Yaskawa INFORM job: apremTRJ4.JBI

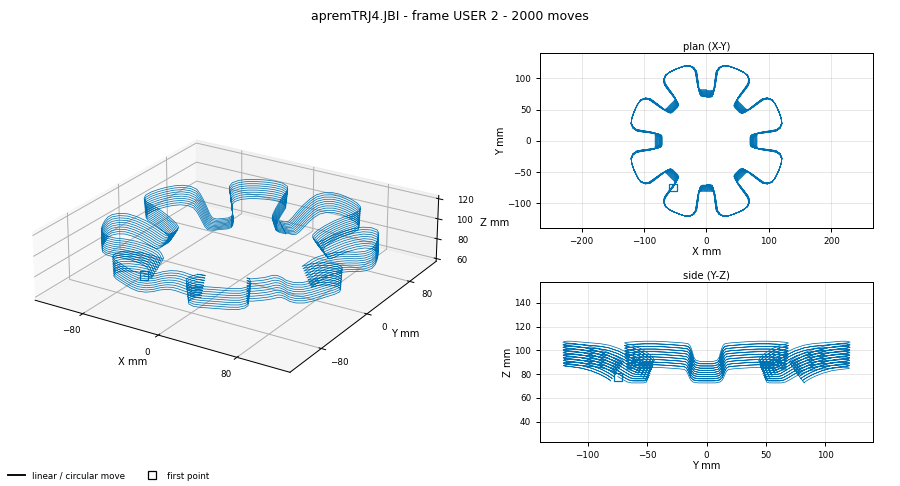
[picture p0: tool path of apremTRJ4.JBI in frame USER 2, 2000 of 2000 moves have a stored position in this frame; points joined in program order, loops and branches not executed]
/JOB
//NAME apremTRJ4
//POS
///NPOS 2000,0,0,0,0,0
///USER 2
///TOOL 1
///POSTYPE USER
///RECTAN
///RCONF 1,0,0,0,0,0,0,0,0,0,0,0,0,0,0,0,0,0,0,0,0,0,0,0
C00000=-53.765,-74.632,78.012,177.9395,-3.2342,0.0000
C00001=-51.010,-70.134,75.345,-179.2635,1.4013,0.0000
C00002=-50.421,-66.568,73.433,174.4013,27.1844,0.0000
C00003=-52.955,-63.098,72.678,152.6245,29.3823,0.0000
C00004=-55.786,-60.507,72.646,149.9913,27.7136,0.0000
C00005=-58.192,-58.192,72.667,151.1075,28.8919,0.0000
C00006=-60.507,-55.786,72.646,152.2867,30.0091,0.0000
C00007=-63.099,-52.955,72.678,150.6167,27.3735,0.0000
C00008=-66.568,-50.421,73.433,152.8156,5.5988,0.0000
C00009=-70.134,-51.010,75.345,178.5987,-0.7365,0.0000
C00010=-74.632,-53.765,78.012,-176.7658,2.0605,0.0000
C00011=-80.322,-57.816,80.784,-174.8040,3.4978,0.0000
C00012=-86.699,-62.416,82.923,-173.5056,4.3301,0.0000
C00013=-92.902,-66.405,83.982,-172.7331,2.9843,0.0000
C00014=-99.586,-67.141,84.541,-175.1721,-0.8383,0.0000
C00015=-105.834,-64.370,84.996,-178.0904,-1.4950,0.0000
C00016=-110.354,-58.600,85.456,-179.9251,-0.1383,0.0000
C00017=-113.876,-51.533,85.759,-179.9922,-0.0171,0.0000
C00018=-116.962,-44.084,85.759,-179.9934,-0.0176,0.0000
C00019=-119.469,-36.595,85.456,-179.9552,-0.1508,0.0000
C00020=-120.352,-29.319,84.996,179.7066,-2.4067,0.0000
C00021=-117.894,-22.942,84.541,177.1732,-4.0082,0.0000
C00022=-112.647,-18.736,83.982,172.7605,-3.0512,0.0000
C00023=-105.440,-17.170,82.923,172.3659,-1.5439,0.0000
C00024=-97.679,-15.914,80.784,173.8630,-1.2077,0.0000
C00025=-90.790,-14.755,78.012,176.2584,-0.8317,0.0000
C00026=-85.662,-13.522,75.345,-178.4885,0.4702,0.0000
C00027=-82.723,-11.418,73.433,-163.6249,23.3873,0.0000
C00028=-82.062,-7.172,72.678,-178.1671,37.3904,0.0000
C00029=-82.232,-3.338,72.646,177.8846,37.9487,0.0000
C00030=-82.296,0.000,72.667,179.9994,37.9698,0.0000
C00031=-82.232,3.338,72.646,-177.8840,37.9488,0.0000
C00032=-82.062,7.172,72.678,178.1644,37.3898,0.0000
C00033=-82.723,11.418,73.433,163.6250,23.3874,0.0000
C00034=-85.662,13.522,75.345,178.4885,0.4702,0.0000
C00035=-90.790,14.755,78.012,-176.2584,-0.8317,0.0000
C00036=-97.679,15.914,80.784,-173.8630,-1.2077,0.0000
C00037=-105.440,17.170,82.923,-172.3659,-1.5439,0.0000
C00038=-112.647,18.736,83.982,-172.7605,-3.0512,0.0000
C00039=-117.894,22.942,84.541,-177.1732,-4.0082,0.0000
C00040=-120.352,29.319,84.996,-179.7066,-2.4067,0.0000
C00041=-119.469,36.595,85.456,179.9552,-0.1508,0.0000
C00042=-116.962,44.084,85.759,179.9934,-0.0176,0.0000
C00043=-113.876,51.533,85.759,179.9922,-0.0171,0.0000
C00044=-110.354,58.600,85.456,179.9251,-0.1383,0.0000
C00045=-105.834,64.370,84.996,178.0904,-1.4950,0.0000
C00046=-99.586,67.141,84.541,175.1721,-0.8383,0.0000
C00047=-92.902,66.405,83.982,172.7331,2.9843,0.0000
C00048=-86.699,62.416,82.923,173.5056,4.3301,0.0000
C00049=-80.322,57.816,80.784,174.8040,3.4978,0.0000
C00050=-74.632,53.765,78.012,176.7658,2.0605,0.0000
C00051=-70.134,51.010,75.345,-178.5987,-0.7365,0.0000
C00052=-66.568,50.421,73.433,-152.8156,5.5987,0.0000
C00053=-63.098,52.955,72.678,-150.6177,27.3755,0.0000
C00054=-60.507,55.786,72.646,-152.2864,30.0087,0.0000
C00055=-58.192,58.192,72.667,-151.1081,28.8925,0.0000
C00056=-55.786,60.507,72.646,-149.9909,27.7133,0.0000
C00057=-52.955,63.099,72.678,-152.6265,29.3833,0.0000
C00058=-50.421,66.568,73.433,-174.4012,27.1844,0.0000
C00059=-51.010,70.134,75.345,179.2635,1.4013,0.0000
C00060=-53.765,74.632,78.012,-177.9395,-3.2342,0.0000
C00061=-57.816,80.322,80.784,-176.5022,-5.1960,0.0000
C00062=-62.416,86.699,82.923,-175.6699,-6.4944,0.0000
C00063=-66.405,92.902,83.982,-177.0157,-7.2669,0.0000
C00064=-67.141,99.586,84.541,179.1617,-4.8279,0.0000
C00065=-64.370,105.834,84.996,178.5050,-1.9096,0.0000
C00066=-58.600,110.354,85.456,179.8617,-0.0749,0.0000
C00067=-51.533,113.876,85.759,179.9829,-0.0078,0.0000
C00068=-44.084,116.962,85.759,179.9824,-0.0066,0.0000
C00069=-36.595,119.469,85.456,179.8492,-0.0448,0.0000
C00070=-29.319,120.352,84.996,177.5933,0.2934,0.0000
C00071=-22.942,117.894,84.541,175.9918,2.8268,0.0000
C00072=-18.736,112.647,83.982,176.9488,7.2395,0.0000
C00073=-17.170,105.440,82.923,178.4561,7.6341,0.0000
C00074=-15.914,97.679,80.784,178.7923,6.1370,0.0000
C00075=-14.755,90.790,78.012,179.1683,3.7416,0.0000
C00076=-13.522,85.662,75.345,-179.5298,-1.5115,0.0000
C00077=-11.418,82.723,73.433,-156.6126,-16.3750,0.0000
C00078=-7.172,82.062,72.678,-142.6102,-1.8356,0.0000
C00079=-3.338,82.232,72.646,-142.0512,2.1160,0.0000
C00080=0.000,82.296,72.667,-142.0302,-0.0006,0.0000
C00081=0.000,80.948,74.406,-142.4252,-0.0006,0.0000
C00082=3.215,80.888,74.384,-142.4452,-2.0536,0.0000
C00083=6.965,80.731,74.417,-143.0509,2.1075,0.0000
C00084=11.165,81.441,75.203,-157.7434,16.2795,0.0000
C00085=13.215,84.505,77.191,-179.7323,0.9131,0.0000
C00086=14.409,89.830,79.960,179.1649,-3.9269,0.0000
C00087=15.548,96.964,82.833,178.8415,-6.1204,0.0000
C00088=16.788,104.985,85.041,178.5474,-7.5066,0.0000
C00089=18.327,112.424,86.132,177.1014,-7.1283,0.0000
C00090=22.561,117.848,86.707,176.0893,-2.8270,0.0000
C00091=29.019,120.407,87.175,177.6414,-0.3022,0.0000
C00092=36.407,119.531,87.647,179.8514,0.0441,0.0000
C00093=44.020,116.986,87.958,179.9827,0.0065,0.0000
C00094=51.595,113.849,87.958,179.9832,0.0077,0.0000
C00095=58.777,110.265,87.647,179.8638,0.0739,0.0000
C00096=64.621,105.660,87.175,178.5453,1.8817,0.0000
C00097=67.378,99.284,86.707,179.2311,4.7592,0.0000
C00098=66.537,92.455,86.132,-176.9875,7.0817,0.0000
C00099=62.365,86.107,85.041,-175.6969,6.3399,0.0000
C00100=57.570,79.558,82.833,-176.4794,5.1497,0.0000
C00101=53.330,73.708,79.960,-177.8105,3.3677,0.0000
C00102=50.409,69.099,77.191,179.5436,-0.8349,0.0000
C00103=49.693,65.482,75.203,-175.2620,-26.3759,0.0000
C00104=52.161,62.011,74.417,-153.1680,-29.1562,0.0000
C00105=54.923,59.470,74.384,-150.3596,-27.3978,0.0000
C00106=57.239,57.239,74.406,-151.4512,-28.5481,0.0000
C00107=59.470,54.923,74.384,-152.6025,-29.6408,0.0000
C00108=62.011,52.160,74.417,-150.8427,-26.8300,0.0000
C00109=65.482,49.693,75.203,-153.6242,-4.7380,0.0000
C00110=69.099,50.409,77.191,-179.1651,0.4564,0.0000
C00111=73.708,53.330,79.960,176.6323,-2.1895,0.0000
C00112=79.558,57.570,82.833,174.8503,-3.5206,0.0000
C00113=86.107,62.365,85.041,173.6601,-4.3031,0.0000
C00114=92.455,66.537,86.132,172.9183,-3.0125,0.0000
C00115=99.284,67.378,86.707,175.2408,0.7689,0.0000
C00116=105.660,64.621,87.175,178.1183,1.4547,0.0000
C00117=110.265,58.777,87.647,179.9261,0.1362,0.0000
C00118=113.849,51.595,87.958,179.9923,0.0168,0.0000
C00119=116.986,44.020,87.958,179.9935,0.0173,0.0000
C00120=119.531,36.407,87.647,179.9559,0.1486,0.0000
C00121=120.407,29.019,87.175,-179.6978,2.3586,0.0000
C00122=117.848,22.561,86.707,-177.1730,3.9107,0.0000
C00123=112.424,18.327,86.132,-172.8717,2.8986,0.0000
C00124=104.985,16.788,85.041,-172.4934,1.4526,0.0000
C00125=96.964,15.548,82.833,-173.8796,1.1585,0.0000
C00126=89.830,14.409,79.960,-176.0731,0.8351,0.0000
C00127=84.505,13.215,77.191,179.0869,-0.2677,0.0000
C00128=81.441,11.165,75.203,163.7205,-22.2566,0.0000
C00129=80.731,6.965,74.417,177.8925,-36.9491,0.0000
C00130=80.888,3.215,74.384,-177.9464,-37.5548,0.0000
C00131=80.948,0.000,74.406,-179.9994,-37.5748,0.0000
C00132=80.888,-3.215,74.384,177.9457,-37.5548,0.0000
C00133=80.731,-6.965,74.417,-177.8898,-36.9485,0.0000
C00134=81.441,-11.165,75.203,-163.7205,-22.2566,0.0000
C00135=84.505,-13.215,77.191,-179.0869,-0.2677,0.0000
C00136=89.830,-14.409,79.960,176.0731,0.8351,0.0000
C00137=96.964,-15.548,82.833,173.8796,1.1585,0.0000
C00138=104.985,-16.788,85.041,172.4934,1.4526,0.0000
C00139=112.424,-18.327,86.132,172.8717,2.8986,0.0000
C00140=117.848,-22.561,86.707,177.1730,3.9107,0.0000
C00141=120.407,-29.019,87.175,179.6978,2.3586,0.0000
C00142=119.531,-36.407,87.647,-179.9559,0.1486,0.0000
C00143=116.986,-44.020,87.958,-179.9935,0.0173,0.0000
C00144=113.849,-51.595,87.958,-179.9923,0.0168,0.0000
C00145=110.265,-58.777,87.647,-179.9261,0.1362,0.0000
C00146=105.660,-64.621,87.175,-178.1183,1.4547,0.0000
C00147=99.284,-67.378,86.707,-175.2408,0.7689,0.0000
C00148=92.455,-66.537,86.132,-172.9183,-3.0125,0.0000
C00149=86.107,-62.365,85.041,-173.6601,-4.3031,0.0000
C00150=79.558,-57.570,82.833,-174.8503,-3.5206,0.0000
C00151=73.708,-53.330,79.960,-176.6323,-2.1895,0.0000
C00152=69.099,-50.409,77.191,179.1651,0.4564,0.0000
C00153=65.482,-49.693,75.203,153.6241,-4.7380,0.0000
C00154=62.011,-52.161,74.417,150.8438,-26.8320,0.0000
C00155=59.470,-54.923,74.384,152.6022,-29.6404,0.0000
C00156=57.239,-57.239,74.406,151.4519,-28.5488,0.0000
C00157=54.923,-59.470,74.384,150.3592,-27.3975,0.0000
C00158=52.160,-62.011,74.417,153.1700,-29.1573,0.0000
C00159=49.693,-65.482,75.203,175.2620,-26.3758,0.0000
C00160=50.409,-69.099,77.191,-179.5436,-0.8349,0.0000
C00161=53.330,-73.708,79.960,177.8105,3.3677,0.0000
C00162=57.570,-79.558,82.833,176.4794,5.1497,0.0000
C00163=62.365,-86.107,85.041,175.6969,6.3399,0.0000
C00164=66.537,-92.455,86.132,176.9875,7.0817,0.0000
C00165=67.378,-99.284,86.707,-179.2311,4.7592,0.0000
C00166=64.621,-105.660,87.175,-178.5453,1.8817,0.0000
C00167=58.777,-110.265,87.647,-179.8638,0.0739,0.0000
C00168=51.595,-113.849,87.958,-179.9832,0.0077,0.0000
C00169=44.020,-116.986,87.958,-179.9827,0.0065,0.0000
C00170=36.407,-119.531,87.647,-179.8514,0.0441,0.0000
C00171=29.019,-120.407,87.175,-177.6414,-0.3022,0.0000
C00172=22.561,-117.848,86.707,-176.0893,-2.8270,0.0000
C00173=18.327,-112.424,86.132,-177.1014,-7.1283,0.0000
C00174=16.788,-104.985,85.041,-178.5474,-7.5066,0.0000
C00175=15.548,-96.964,82.833,-178.8415,-6.1204,0.0000
C00176=14.409,-89.830,79.960,-179.1649,-3.9269,0.0000
C00177=13.215,-84.505,77.191,179.7323,0.9131,0.0000
C00178=11.165,-81.441,75.203,157.7434,16.2795,0.0000
C00179=6.965,-80.731,74.417,143.0509,2.1075,0.0000
C00180=3.215,-80.888,74.384,142.4452,-2.0536,0.0000
C00181=0.000,-80.948,74.406,142.4252,-0.0006,0.0000
C00182=0.000,-80.948,74.406,142.4252,-0.0006,0.0000
C00183=-3.215,-80.888,74.384,142.4452,2.0543,0.0000
C00184=-6.965,-80.731,74.417,143.0515,-2.1102,0.0000
C00185=-11.165,-81.441,75.203,157.7434,-16.2795,0.0000
C00186=-13.215,-84.505,77.191,179.7323,-0.9131,0.0000
C00187=-14.409,-89.830,79.960,-179.1649,3.9269,0.0000
C00188=-15.548,-96.964,82.833,-178.8415,6.1204,0.0000
C00189=-16.788,-104.985,85.041,-178.5474,7.5066,0.0000
C00190=-18.327,-112.424,86.132,-177.1014,7.1283,0.0000
C00191=-22.561,-117.848,86.707,-176.0893,2.8270,0.0000
C00192=-29.019,-120.407,87.175,-177.6414,0.3022,0.0000
C00193=-36.407,-119.531,87.647,-179.8514,-0.0441,0.0000
C00194=-44.020,-116.986,87.958,-179.9827,-0.0065,0.0000
C00195=-51.595,-113.849,87.958,-179.9832,-0.0077,0.0000
C00196=-58.777,-110.265,87.647,-179.8638,-0.0739,0.0000
C00197=-64.621,-105.660,87.175,-178.5453,-1.8817,0.0000
C00198=-67.378,-99.284,86.707,-179.2311,-4.7592,0.0000
C00199=-66.537,-92.455,86.132,176.9875,-7.0817,0.0000
C00200=-62.365,-86.107,85.041,175.6969,-6.3399,0.0000
C00201=-57.570,-79.558,82.833,176.4794,-5.1497,0.0000
C00202=-53.330,-73.708,79.960,177.8105,-3.3677,0.0000
C00203=-50.409,-69.099,77.191,-179.5436,0.8349,0.0000
C00204=-49.693,-65.482,75.203,175.2620,26.3759,0.0000
C00205=-52.161,-62.011,74.417,153.1680,29.1562,0.0000
C00206=-54.923,-59.470,74.384,150.3596,27.3978,0.0000
C00207=-57.239,-57.239,74.406,151.4512,28.5481,0.0000
C00208=-59.470,-54.923,74.384,152.6025,29.6408,0.0000
C00209=-62.011,-52.160,74.417,150.8427,26.8300,0.0000
C00210=-65.482,-49.693,75.203,153.6242,4.7380,0.0000
C00211=-69.099,-50.409,77.191,179.1651,-0.4564,0.0000
C00212=-73.708,-53.330,79.960,-176.6323,2.1895,0.0000
C00213=-79.558,-57.570,82.833,-174.8503,3.5206,0.0000
C00214=-86.107,-62.365,85.041,-173.6601,4.3031,0.0000
C00215=-92.455,-66.537,86.132,-172.9183,3.0125,0.0000
C00216=-99.284,-67.378,86.707,-175.2408,-0.7689,0.0000
C00217=-105.660,-64.621,87.175,-178.1183,-1.4547,0.0000
C00218=-110.265,-58.777,87.647,-179.9261,-0.1362,0.0000
C00219=-113.849,-51.595,87.958,-179.9923,-0.0168,0.0000
C00220=-116.986,-44.020,87.958,-179.9935,-0.0173,0.0000
C00221=-119.531,-36.407,87.647,-179.9559,-0.1486,0.0000
C00222=-120.407,-29.019,87.175,179.6978,-2.3586,0.0000
C00223=-117.848,-22.561,86.707,177.1730,-3.9107,0.0000
C00224=-112.424,-18.327,86.132,172.8717,-2.8986,0.0000
C00225=-104.985,-16.788,85.041,172.4934,-1.4526,0.0000
C00226=-96.964,-15.548,82.833,173.8796,-1.1585,0.0000
C00227=-89.830,-14.409,79.960,176.0731,-0.8351,0.0000
C00228=-84.505,-13.215,77.191,-179.0869,0.2677,0.0000
C00229=-81.441,-11.165,75.203,-163.7205,22.2566,0.0000
C00230=-80.731,-6.965,74.417,-177.8925,36.9491,0.0000
C00231=-80.888,-3.215,74.384,177.9464,37.5548,0.0000
C00232=-80.948,0.000,74.406,179.9994,37.5748,0.0000
C00233=-80.888,3.215,74.384,-177.9457,37.5548,0.0000
C00234=-80.731,6.965,74.417,177.8898,36.9485,0.0000
C00235=-81.441,11.165,75.203,163.7205,22.2566,0.0000
C00236=-84.505,13.215,77.191,179.0869,0.2677,0.0000
C00237=-89.830,14.409,79.960,-176.0731,-0.8351,0.0000
C00238=-96.964,15.548,82.833,-173.8796,-1.1585,0.0000
C00239=-104.985,16.788,85.041,-172.4934,-1.4526,0.0000
C00240=-112.424,18.327,86.132,-172.8717,-2.8986,0.0000
C00241=-117.848,22.561,86.707,-177.1730,-3.9107,0.0000
C00242=-120.407,29.019,87.175,-179.6978,-2.3586,0.0000
C00243=-119.531,36.407,87.647,179.9559,-0.1486,0.0000
C00244=-116.986,44.020,87.958,179.9935,-0.0173,0.0000
C00245=-113.849,51.595,87.958,179.9923,-0.0168,0.0000
C00246=-110.265,58.777,87.647,179.9261,-0.1362,0.0000
C00247=-105.660,64.621,87.175,178.1183,-1.4547,0.0000
C00248=-99.284,67.378,86.707,175.2408,-0.7689,0.0000
C00249=-92.455,66.537,86.132,172.9183,3.0125,0.0000
C00250=-86.107,62.365,85.041,173.6601,4.3031,0.0000
C00251=-79.558,57.570,82.833,174.8503,3.5206,0.0000
C00252=-73.708,53.330,79.960,176.6323,2.1895,0.0000
C00253=-69.099,50.409,77.191,-179.1651,-0.4564,0.0000
C00254=-65.482,49.693,75.203,-153.6241,4.7380,0.0000
C00255=-62.011,52.161,74.417,-150.8438,26.8320,0.0000
C00256=-59.470,54.923,74.384,-152.6022,29.6404,0.0000
C00257=-57.239,57.239,74.406,-151.4519,28.5488,0.0000
C00258=-54.923,59.470,74.384,-150.3592,27.3975,0.0000
C00259=-52.160,62.011,74.417,-153.1700,29.1573,0.0000
C00260=-49.693,65.482,75.203,-175.2620,26.3758,0.0000
C00261=-50.409,69.099,77.191,179.5436,0.8349,0.0000
C00262=-53.330,73.708,79.960,-177.8105,-3.3677,0.0000
C00263=-57.570,79.558,82.833,-176.4794,-5.1497,0.0000
C00264=-62.365,86.107,85.041,-175.6969,-6.3399,0.0000
C00265=-66.537,92.455,86.132,-176.9875,-7.0817,0.0000
C00266=-67.378,99.284,86.707,179.2311,-4.7592,0.0000
C00267=-64.621,105.660,87.175,178.5453,-1.8817,0.0000
C00268=-58.777,110.265,87.647,179.8638,-0.0739,0.0000
C00269=-51.595,113.849,87.958,179.9832,-0.0077,0.0000
C00270=-44.020,116.986,87.958,179.9827,-0.0065,0.0000
C00271=-36.407,119.531,87.647,179.8514,-0.0441,0.0000
C00272=-29.019,120.407,87.175,177.6414,0.3022,0.0000
C00273=-22.561,117.848,86.707,176.0893,2.8270,0.0000
C00274=-18.327,112.424,86.132,177.1014,7.1283,0.0000
C00275=-16.788,104.985,85.041,178.5474,7.5066,0.0000
C00276=-15.548,96.964,82.833,178.8415,6.1204,0.0000
C00277=-14.409,89.830,79.960,179.1649,3.9269,0.0000
C00278=-13.215,84.505,77.191,-179.7323,-0.9131,0.0000
C00279=-11.165,81.441,75.203,-157.7434,-16.2795,0.0000
C00280=-6.965,80.731,74.417,-143.0515,-2.1102,0.0000
C00281=-3.215,80.888,74.384,-142.4452,2.0543,0.0000
C00282=0.000,80.948,74.406,-142.4252,-0.0006,0.0000
C00283=0.000,79.613,76.155,-142.8783,-0.0007,0.0000
C00284=3.093,79.558,76.131,-142.8972,-1.9868,0.0000
C00285=6.760,79.413,76.167,-143.5531,2.3727,0.0000
C00286=10.915,80.173,76.983,-158.8902,16.1064,0.0000
C00287=12.913,83.364,79.048,-179.8982,0.3680,0.0000
C00288=14.070,88.888,81.919,179.1707,-4.0693,0.0000
C00289=15.193,96.269,84.889,178.8939,-6.0643,0.0000
C00290=16.419,104.545,87.165,178.6389,-7.3362,0.0000
C00291=17.933,112.210,88.285,177.2596,-6.9702,0.0000
C00292=22.194,117.804,88.875,176.2095,-2.8032,0.0000
C00293=28.731,120.459,89.355,177.7041,-0.3075,0.0000
C00294=36.227,119.590,89.839,179.8547,0.0430,0.0000
C00295=43.959,117.010,90.157,179.9831,0.0063,0.0000
C00296=51.654,113.822,90.157,179.9836,0.0075,0.0000
C00297=58.947,110.179,89.839,179.8669,0.0724,0.0000
C00298=64.862,105.493,89.355,178.5934,1.8411,0.0000
C00299=67.607,98.993,88.875,179.2995,4.6577,0.0000
C00300=66.664,92.025,88.285,-176.9888,6.8594,0.0000
C00301=62.315,85.535,87.165,-175.7544,6.1549,0.0000
C00302=57.329,78.815,84.889,-176.4825,5.0731,0.0000
C00303=52.904,72.802,81.919,-177.7054,3.4644,0.0000
C00304=49.817,68.078,79.048,179.8118,-0.3322,0.0000
C00305=48.973,64.408,76.983,-176.0638,-25.5091,0.0000
C00306=51.374,60.933,76.167,-153.7604,-28.8775,0.0000
C00307=54.069,58.443,76.131,-150.7789,-27.0355,0.0000
C00308=56.295,56.295,76.155,-151.8438,-28.1554,0.0000
C00309=58.443,54.069,76.131,-152.9649,-29.2216,0.0000
C00310=60.934,51.373,76.167,-151.1215,-26.2375,0.0000
C00311=64.409,48.973,76.983,-154.4910,-3.9361,0.0000
C00312=68.078,49.817,79.048,-179.6678,0.1882,0.0000
C00313=72.802,52.904,81.919,176.5356,-2.2946,0.0000
C00314=78.815,57.329,84.889,174.9269,-3.5175,0.0000
C00315=85.535,62.315,87.165,173.8451,-4.2456,0.0000
C00316=92.025,66.664,88.285,173.1406,-3.0112,0.0000
C00317=98.993,67.607,88.875,175.3423,0.7005,0.0000
C00318=105.493,64.862,89.355,178.1589,1.4066,0.0000
C00319=110.179,58.947,89.839,179.9276,0.1331,0.0000
C00320=113.822,51.654,90.157,179.9925,0.0164,0.0000
C00321=117.010,43.959,90.157,179.9937,0.0169,0.0000
C00322=119.590,36.227,89.839,179.9570,0.1453,0.0000
C00323=120.459,28.731,89.355,-179.6925,2.2959,0.0000
C00324=117.804,22.194,88.875,-177.1968,3.7905,0.0000
C00325=112.210,17.933,88.285,-173.0298,2.7404,0.0000
C00326=104.545,16.419,87.165,-172.6638,1.3611,0.0000
C00327=96.269,15.193,84.889,-173.9357,1.1061,0.0000
C00328=88.888,14.070,81.919,-175.9307,0.8293,0.0000
C00329=83.364,12.913,79.048,179.6320,-0.1018,0.0000
C00330=80.173,10.915,76.983,163.8936,-21.1098,0.0000
C00331=79.413,6.760,76.167,177.6273,-36.4469,0.0000
C00332=79.558,3.093,76.131,-178.0132,-37.1028,0.0000
C00333=79.613,0.000,76.155,-179.9993,-37.1217,0.0000
C00334=79.558,-3.093,76.131,178.0125,-37.1029,0.0000
C00335=79.413,-6.760,76.167,-177.6245,-36.4463,0.0000
C00336=80.173,-10.915,76.983,-163.8937,-21.1097,0.0000
C00337=83.364,-12.913,79.048,-179.6320,-0.1018,0.0000
C00338=88.888,-14.070,81.919,175.9307,0.8293,0.0000
C00339=96.269,-15.193,84.889,173.9357,1.1061,0.0000
C00340=104.545,-16.419,87.165,172.6638,1.3611,0.0000
C00341=112.210,-17.933,88.285,173.0298,2.7404,0.0000
C00342=117.804,-22.194,88.875,177.1968,3.7905,0.0000
C00343=120.459,-28.731,89.355,179.6925,2.2959,0.0000
C00344=119.590,-36.227,89.839,-179.9570,0.1453,0.0000
C00345=117.010,-43.959,90.157,-179.9937,0.0169,0.0000
C00346=113.822,-51.654,90.157,-179.9925,0.0164,0.0000
C00347=110.179,-58.947,89.839,-179.9276,0.1331,0.0000
C00348=105.493,-64.862,89.355,-178.1589,1.4066,0.0000
C00349=98.993,-67.607,88.875,-175.3423,0.7005,0.0000
C00350=92.025,-66.664,88.285,-173.1406,-3.0112,0.0000
C00351=85.535,-62.315,87.165,-173.8451,-4.2456,0.0000
C00352=78.815,-57.329,84.889,-174.9269,-3.5175,0.0000
C00353=72.802,-52.904,81.919,-176.5356,-2.2946,0.0000
C00354=68.078,-49.817,79.048,179.6678,0.1882,0.0000
C00355=64.408,-48.973,76.983,154.4909,-3.9362,0.0000
C00356=60.933,-51.374,76.167,151.1225,-26.2396,0.0000
C00357=58.443,-54.069,76.131,152.9645,-29.2211,0.0000
C00358=56.295,-56.295,76.155,151.8446,-28.1562,0.0000
C00359=54.069,-58.443,76.131,150.7784,-27.0351,0.0000
C00360=51.373,-60.934,76.167,153.7625,-28.8785,0.0000
C00361=48.973,-64.409,76.983,176.0639,-25.5090,0.0000
C00362=49.817,-68.078,79.048,-179.8118,-0.3322,0.0000
C00363=52.904,-72.802,81.919,177.7054,3.4644,0.0000
C00364=57.329,-78.815,84.889,176.4825,5.0731,0.0000
C00365=62.315,-85.535,87.165,175.7544,6.1549,0.0000
C00366=66.664,-92.025,88.285,176.9888,6.8594,0.0000
C00367=67.607,-98.993,88.875,-179.2995,4.6577,0.0000
C00368=64.862,-105.493,89.355,-178.5934,1.8411,0.0000
C00369=58.947,-110.179,89.839,-179.8669,0.0724,0.0000
C00370=51.654,-113.822,90.157,-179.9836,0.0075,0.0000
C00371=43.959,-117.010,90.157,-179.9831,0.0063,0.0000
C00372=36.227,-119.590,89.839,-179.8547,0.0430,0.0000
C00373=28.731,-120.459,89.355,-177.7041,-0.3075,0.0000
C00374=22.194,-117.804,88.875,-176.2095,-2.8032,0.0000
C00375=17.933,-112.210,88.285,-177.2596,-6.9702,0.0000
C00376=16.419,-104.545,87.165,-178.6389,-7.3362,0.0000
C00377=15.193,-96.269,84.889,-178.8939,-6.0643,0.0000
C00378=14.070,-88.888,81.919,-179.1707,-4.0693,0.0000
C00379=12.913,-83.364,79.048,179.8982,0.3680,0.0000
C00380=10.915,-80.173,76.983,158.8902,16.1064,0.0000
C00381=6.760,-79.413,76.167,143.5531,2.3727,0.0000
C00382=3.093,-79.558,76.131,142.8972,-1.9868,0.0000
C00383=0.000,-79.613,76.155,142.8783,-0.0007,0.0000
C00384=0.000,-79.613,76.155,142.8783,-0.0007,0.0000
C00385=-3.093,-79.558,76.131,142.8971,1.9875,0.0000
C00386=-6.760,-79.413,76.167,143.5537,-2.3755,0.0000
C00387=-10.915,-80.173,76.983,158.8903,-16.1063,0.0000
C00388=-12.913,-83.364,79.048,179.8982,-0.3680,0.0000
C00389=-14.070,-88.888,81.919,-179.1707,4.0693,0.0000
C00390=-15.193,-96.269,84.889,-178.8939,6.0643,0.0000
C00391=-16.419,-104.545,87.165,-178.6389,7.3362,0.0000
C00392=-17.933,-112.210,88.285,-177.2596,6.9702,0.0000
C00393=-22.194,-117.804,88.875,-176.2095,2.8032,0.0000
C00394=-28.731,-120.459,89.355,-177.7041,0.3075,0.0000
C00395=-36.227,-119.590,89.839,-179.8547,-0.0430,0.0000
C00396=-43.959,-117.010,90.157,-179.9831,-0.0063,0.0000
C00397=-51.654,-113.822,90.157,-179.9836,-0.0075,0.0000
C00398=-58.947,-110.179,89.839,-179.8669,-0.0724,0.0000
C00399=-64.862,-105.493,89.355,-178.5934,-1.8411,0.0000
C00400=-67.607,-98.993,88.875,-179.2995,-4.6577,0.0000
C00401=-66.664,-92.025,88.285,176.9888,-6.8594,0.0000
C00402=-62.315,-85.535,87.165,175.7544,-6.1549,0.0000
C00403=-57.329,-78.815,84.889,176.4825,-5.0731,0.0000
C00404=-52.904,-72.802,81.919,177.7054,-3.4644,0.0000
C00405=-49.817,-68.078,79.048,-179.8118,0.3322,0.0000
C00406=-48.973,-64.408,76.983,176.0638,25.5091,0.0000
C00407=-51.374,-60.933,76.167,153.7604,28.8775,0.0000
C00408=-54.069,-58.443,76.131,150.7789,27.0355,0.0000
C00409=-56.295,-56.295,76.155,151.8438,28.1554,0.0000
C00410=-58.443,-54.069,76.131,152.9649,29.2216,0.0000
C00411=-60.934,-51.373,76.167,151.1215,26.2375,0.0000
C00412=-64.409,-48.973,76.983,154.4910,3.9361,0.0000
C00413=-68.078,-49.817,79.048,179.6678,-0.1882,0.0000
C00414=-72.802,-52.904,81.919,-176.5356,2.2946,0.0000
C00415=-78.815,-57.329,84.889,-174.9269,3.5175,0.0000
C00416=-85.535,-62.315,87.165,-173.8451,4.2456,0.0000
C00417=-92.025,-66.664,88.285,-173.1406,3.0112,0.0000
C00418=-98.993,-67.607,88.875,-175.3423,-0.7005,0.0000
C00419=-105.493,-64.862,89.355,-178.1589,-1.4066,0.0000
C00420=-110.179,-58.947,89.839,-179.9276,-0.1331,0.0000
C00421=-113.822,-51.654,90.157,-179.9925,-0.0164,0.0000
C00422=-117.010,-43.959,90.157,-179.9937,-0.0169,0.0000
C00423=-119.590,-36.227,89.839,-179.9570,-0.1453,0.0000
C00424=-120.459,-28.731,89.355,179.6925,-2.2959,0.0000
C00425=-117.804,-22.194,88.875,177.1968,-3.7905,0.0000
C00426=-112.210,-17.933,88.285,173.0298,-2.7404,0.0000
C00427=-104.545,-16.419,87.165,172.6638,-1.3611,0.0000
C00428=-96.269,-15.193,84.889,173.9357,-1.1061,0.0000
C00429=-88.888,-14.070,81.919,175.9307,-0.8293,0.0000
C00430=-83.364,-12.913,79.048,-179.6320,0.1018,0.0000
C00431=-80.173,-10.915,76.983,-163.8936,21.1098,0.0000
C00432=-79.413,-6.760,76.167,-177.6273,36.4469,0.0000
C00433=-79.558,-3.093,76.131,178.0132,37.1028,0.0000
C00434=-79.613,0.000,76.155,179.9993,37.1217,0.0000
C00435=-79.558,3.093,76.131,-178.0125,37.1029,0.0000
C00436=-79.413,6.760,76.167,177.6245,36.4463,0.0000
C00437=-80.173,10.915,76.983,163.8937,21.1097,0.0000
C00438=-83.364,12.913,79.048,179.6320,0.1018,0.0000
C00439=-88.888,14.070,81.919,-175.9307,-0.8293,0.0000
C00440=-96.269,15.193,84.889,-173.9357,-1.1061,0.0000
C00441=-104.545,16.419,87.165,-172.6638,-1.3611,0.0000
C00442=-112.210,17.933,88.285,-173.0298,-2.7404,0.0000
C00443=-117.804,22.194,88.875,-177.1968,-3.7905,0.0000
C00444=-120.459,28.731,89.355,-179.6925,-2.2959,0.0000
C00445=-119.590,36.227,89.839,179.9570,-0.1453,0.0000
C00446=-117.010,43.959,90.157,179.9937,-0.0169,0.0000
C00447=-113.822,51.654,90.157,179.9925,-0.0164,0.0000
C00448=-110.179,58.947,89.839,179.9276,-0.1331,0.0000
C00449=-105.493,64.862,89.355,178.1589,-1.4066,0.0000
C00450=-98.993,67.607,88.875,175.3423,-0.7005,0.0000
C00451=-92.025,66.664,88.285,173.1406,3.0112,0.0000
C00452=-85.535,62.315,87.165,173.8451,4.2456,0.0000
C00453=-78.815,57.329,84.889,174.9269,3.5175,0.0000
C00454=-72.802,52.904,81.919,176.5356,2.2946,0.0000
C00455=-68.078,49.817,79.048,-179.6678,-0.1882,0.0000
C00456=-64.408,48.973,76.983,-154.4909,3.9362,0.0000
C00457=-60.933,51.374,76.167,-151.1225,26.2396,0.0000
C00458=-58.443,54.069,76.131,-152.9645,29.2211,0.0000
C00459=-56.295,56.295,76.155,-151.8446,28.1562,0.0000
C00460=-54.069,58.443,76.131,-150.7784,27.0351,0.0000
C00461=-51.373,60.934,76.167,-153.7625,28.8785,0.0000
C00462=-48.973,64.409,76.983,-176.0639,25.5090,0.0000
C00463=-49.817,68.078,79.048,179.8118,0.3322,0.0000
C00464=-52.904,72.802,81.919,-177.7054,-3.4644,0.0000
C00465=-57.329,78.815,84.889,-176.4825,-5.0731,0.0000
C00466=-62.315,85.535,87.165,-175.7544,-6.1549,0.0000
C00467=-66.664,92.025,88.285,-176.9888,-6.8594,0.0000
C00468=-67.607,98.993,88.875,179.2995,-4.6577,0.0000
C00469=-64.862,105.493,89.355,178.5934,-1.8411,0.0000
C00470=-58.947,110.179,89.839,179.8669,-0.0724,0.0000
C00471=-51.654,113.822,90.157,179.9836,-0.0075,0.0000
C00472=-43.959,117.010,90.157,179.9831,-0.0063,0.0000
C00473=-36.227,119.590,89.839,179.8547,-0.0430,0.0000
C00474=-28.731,120.459,89.355,177.7041,0.3075,0.0000
C00475=-22.194,117.804,88.875,176.2095,2.8032,0.0000
C00476=-17.933,112.210,88.285,177.2596,6.9702,0.0000
C00477=-16.419,104.545,87.165,178.6389,7.3362,0.0000
C00478=-15.193,96.269,84.889,178.8939,6.0643,0.0000
C00479=-14.070,88.888,81.919,179.1707,4.0693,0.0000
C00480=-12.913,83.364,79.048,-179.8982,-0.3680,0.0000
C00481=-10.915,80.173,76.983,-158.8903,-16.1063,0.0000
C00482=-6.760,79.413,76.167,-143.5537,-2.3755,0.0000
C00483=-3.093,79.558,76.131,-142.8971,1.9875,0.0000
C00484=0.000,79.613,76.155,-142.8783,-0.0007,0.0000
C00485=0.000,78.293,77.915,-143.3925,-0.0008,0.0000
C00486=2.973,78.242,77.891,-143.4103,-1.9151,0.0000
C00487=6.557,78.109,77.927,-144.1191,2.6261,0.0000
C00488=10.667,78.920,78.774,-160.0460,15.8589,0.0000
C00489=12.615,82.242,80.917,179.9678,-0.1232,0.0000
C00490=13.739,87.966,83.889,179.1844,-4.1696,0.0000
C00491=14.847,95.594,86.955,178.9489,-5.9694,0.0000
C00492=16.063,104.122,89.294,178.7302,-7.1239,0.0000
C00493=17.555,112.004,90.443,177.4226,-6.7663,0.0000
C00494=21.842,117.762,91.047,176.3515,-2.7551,0.0000
C00495=28.456,120.509,91.537,177.7813,-0.3092,0.0000
C00496=36.055,119.647,92.031,179.8591,0.0416,0.0000
C00497=43.902,117.032,92.356,179.9837,0.0061,0.0000
C00498=51.711,113.797,92.356,179.9842,0.0072,0.0000
C00499=59.109,110.098,92.031,179.8710,0.0703,0.0000
C00500=65.092,105.334,91.537,178.6493,1.7877,0.0000
C00501=67.825,98.715,91.047,179.3663,4.5236,0.0000
C00502=66.785,91.612,90.443,-177.0196,6.6012,0.0000
C00503=62.267,84.984,89.294,-175.8419,5.9402,0.0000
C00504=57.097,78.094,86.955,-176.5113,4.9672,0.0000
C00505=52.487,71.917,83.889,-177.6245,3.5258,0.0000
C00506=49.233,67.074,80.917,-179.9356,0.1099,0.0000
C00507=48.262,63.348,78.774,-176.8035,-24.5888,0.0000
C00508=50.595,59.868,77.927,-154.4024,-28.5432,0.0000
C00509=53.224,57.428,77.891,-151.2512,-26.6247,0.0000
C00510=55.362,55.362,77.915,-152.2872,-27.7119,0.0000
C00511=57.427,53.224,77.891,-153.3757,-28.7493,0.0000
C00512=59.868,50.595,77.927,-151.4558,-25.5955,0.0000
C00513=63.348,48.262,78.775,-155.4114,-3.1964,0.0000
C00514=67.074,49.233,80.917,179.8901,-0.0644,0.0000
C00515=71.917,52.487,83.889,176.4742,-2.3755,0.0000
C00516=78.094,57.097,86.955,175.0328,-3.4887,0.0000
C00517=84.984,62.267,89.294,174.0598,-4.1581,0.0000
C00518=91.612,66.785,90.443,173.3988,-2.9804,0.0000
C00519=98.715,67.825,91.047,175.4764,0.6337,0.0000
C00520=105.334,65.092,91.537,178.2123,1.3507,0.0000
C00521=110.098,59.109,92.031,179.9297,0.1290,0.0000
C00522=113.797,51.711,92.356,179.9928,0.0158,0.0000
C00523=117.032,43.902,92.356,179.9939,0.0163,0.0000
C00524=119.647,36.055,92.031,179.9584,0.1409,0.0000
C00525=120.509,28.456,91.537,-179.6908,2.2187,0.0000
C00526=117.762,21.842,91.047,-177.2449,3.6485,0.0000
C00527=112.004,17.555,90.443,-173.2337,2.5774,0.0000
C00528=104.122,16.063,89.294,-172.8761,1.2698,0.0000
C00529=95.594,14.847,86.955,-174.0306,1.0511,0.0000
C00530=87.966,13.739,83.889,-175.8304,0.8156,0.0000
C00531=82.242,12.615,80.917,-179.8768,0.0322,0.0000
C00532=78.920,10.667,78.774,164.1411,-19.9540,0.0000
C00533=78.109,6.557,77.927,177.3739,-35.8809,0.0000
C00534=78.242,2.973,77.891,-178.0849,-36.5897,0.0000
C00535=78.293,0.000,77.915,-179.9992,-36.6075,0.0000
C00536=78.242,-2.972,77.891,178.0840,-36.5898,0.0000
C00537=78.109,-6.557,77.927,-177.3711,-35.8803,0.0000
C00538=78.920,-10.668,78.775,-164.1412,-19.9538,0.0000
C00539=82.242,-12.615,80.917,179.8768,0.0322,0.0000
C00540=87.966,-13.739,83.889,175.8304,0.8156,0.0000
C00541=95.594,-14.847,86.955,174.0306,1.0511,0.0000
C00542=104.122,-16.063,89.294,172.8761,1.2698,0.0000
C00543=112.004,-17.555,90.443,173.2337,2.5774,0.0000
C00544=117.762,-21.842,91.047,177.2449,3.6485,0.0000
C00545=120.509,-28.456,91.537,179.6908,2.2187,0.0000
C00546=119.647,-36.055,92.031,-179.9584,0.1409,0.0000
C00547=117.032,-43.902,92.356,-179.9939,0.0163,0.0000
C00548=113.797,-51.711,92.356,-179.9928,0.0158,0.0000
C00549=110.098,-59.109,92.031,-179.9297,0.1290,0.0000
C00550=105.334,-65.092,91.537,-178.2123,1.3507,0.0000
C00551=98.715,-67.825,91.047,-175.4764,0.6337,0.0000
C00552=91.612,-66.785,90.443,-173.3988,-2.9804,0.0000
C00553=84.984,-62.267,89.294,-174.0598,-4.1581,0.0000
C00554=78.094,-57.097,86.955,-175.0328,-3.4887,0.0000
C00555=71.917,-52.487,83.889,-176.4742,-2.3755,0.0000
C00556=67.074,-49.233,80.917,-179.8901,-0.0644,0.0000
C00557=63.348,-48.262,78.774,155.4112,-3.1965,0.0000
C00558=59.868,-50.595,77.927,151.4568,-25.5976,0.0000
C00559=57.428,-53.224,77.891,153.3753,-28.7488,0.0000
C00560=55.362,-55.362,77.915,152.2881,-27.7128,0.0000
C00561=53.224,-57.427,77.891,151.2507,-26.6243,0.0000
C00562=50.595,-59.868,77.927,154.4045,-28.5442,0.0000
C00563=48.262,-63.348,78.775,176.8036,-24.5886,0.0000
C00564=49.233,-67.074,80.917,179.9356,0.1099,0.0000
C00565=52.487,-71.917,83.889,177.6245,3.5258,0.0000
C00566=57.097,-78.094,86.955,176.5113,4.9672,0.0000
C00567=62.267,-84.984,89.294,175.8419,5.9402,0.0000
C00568=66.785,-91.612,90.443,177.0196,6.6012,0.0000
C00569=67.825,-98.715,91.047,-179.3663,4.5236,0.0000
C00570=65.092,-105.334,91.537,-178.6493,1.7877,0.0000
C00571=59.109,-110.098,92.031,-179.8710,0.0703,0.0000
C00572=51.711,-113.797,92.356,-179.9842,0.0072,0.0000
C00573=43.902,-117.032,92.356,-179.9837,0.0061,0.0000
C00574=36.055,-119.647,92.031,-179.8591,0.0416,0.0000
C00575=28.456,-120.509,91.537,-177.7813,-0.3092,0.0000
C00576=21.842,-117.762,91.047,-176.3515,-2.7551,0.0000
C00577=17.555,-112.004,90.443,-177.4226,-6.7663,0.0000
C00578=16.063,-104.122,89.294,-178.7302,-7.1239,0.0000
C00579=14.847,-95.594,86.955,-178.9489,-5.9694,0.0000
C00580=13.739,-87.966,83.889,-179.1844,-4.1696,0.0000
C00581=12.615,-82.242,80.917,-179.9678,-0.1232,0.0000
C00582=10.667,-78.920,78.774,160.0460,15.8589,0.0000
C00583=6.557,-78.109,77.927,144.1191,2.6261,0.0000
C00584=2.973,-78.242,77.891,143.4103,-1.9151,0.0000
C00585=0.000,-78.293,77.915,143.3925,-0.0008,0.0000
C00586=0.000,-78.293,77.915,143.3925,-0.0008,0.0000
C00587=-2.972,-78.242,77.891,143.4102,1.9160,0.0000
C00588=-6.557,-78.109,77.927,144.1197,-2.6289,0.0000
C00589=-10.668,-78.920,78.775,160.0462,-15.8588,0.0000
C00590=-12.615,-82.242,80.917,-179.9678,0.1232,0.0000
C00591=-13.739,-87.966,83.889,-179.1844,4.1696,0.0000
C00592=-14.847,-95.594,86.955,-178.9489,5.9694,0.0000
C00593=-16.063,-104.122,89.294,-178.7302,7.1239,0.0000
C00594=-17.555,-112.004,90.443,-177.4226,6.7663,0.0000
C00595=-21.842,-117.762,91.047,-176.3515,2.7551,0.0000
C00596=-28.456,-120.509,91.537,-177.7813,0.3092,0.0000
C00597=-36.055,-119.647,92.031,-179.8591,-0.0416,0.0000
C00598=-43.902,-117.032,92.356,-179.9837,-0.0061,0.0000
C00599=-51.711,-113.797,92.356,-179.9842,-0.0072,0.0000
C00600=-59.109,-110.098,92.031,-179.8710,-0.0703,0.0000
C00601=-65.092,-105.334,91.537,-178.6493,-1.7877,0.0000
C00602=-67.825,-98.715,91.047,-179.3663,-4.5236,0.0000
C00603=-66.785,-91.612,90.443,177.0196,-6.6012,0.0000
C00604=-62.267,-84.984,89.294,175.8419,-5.9402,0.0000
C00605=-57.097,-78.094,86.955,176.5113,-4.9672,0.0000
C00606=-52.487,-71.917,83.889,177.6245,-3.5258,0.0000
C00607=-49.233,-67.074,80.917,179.9356,-0.1099,0.0000
C00608=-48.262,-63.348,78.774,176.8035,24.5888,0.0000
C00609=-50.595,-59.868,77.927,154.4024,28.5432,0.0000
C00610=-53.224,-57.428,77.891,151.2512,26.6247,0.0000
C00611=-55.362,-55.362,77.915,152.2872,27.7119,0.0000
C00612=-57.427,-53.224,77.891,153.3757,28.7493,0.0000
C00613=-59.868,-50.595,77.927,151.4558,25.5955,0.0000
C00614=-63.348,-48.262,78.775,155.4114,3.1964,0.0000
C00615=-67.074,-49.233,80.917,-179.8901,0.0644,0.0000
C00616=-71.917,-52.487,83.889,-176.4742,2.3755,0.0000
C00617=-78.094,-57.097,86.955,-175.0328,3.4887,0.0000
C00618=-84.984,-62.267,89.294,-174.0598,4.1581,0.0000
C00619=-91.612,-66.785,90.443,-173.3988,2.9804,0.0000
C00620=-98.715,-67.825,91.047,-175.4764,-0.6337,0.0000
C00621=-105.334,-65.092,91.537,-178.2123,-1.3507,0.0000
C00622=-110.098,-59.109,92.031,-179.9297,-0.1290,0.0000
C00623=-113.797,-51.711,92.356,-179.9928,-0.0158,0.0000
C00624=-117.032,-43.902,92.356,-179.9939,-0.0163,0.0000
C00625=-119.647,-36.055,92.031,-179.9584,-0.1409,0.0000
C00626=-120.509,-28.456,91.537,179.6908,-2.2187,0.0000
C00627=-117.762,-21.842,91.047,177.2449,-3.6485,0.0000
C00628=-112.004,-17.555,90.443,173.2337,-2.5774,0.0000
C00629=-104.122,-16.063,89.294,172.8761,-1.2698,0.0000
C00630=-95.594,-14.847,86.955,174.0306,-1.0511,0.0000
C00631=-87.966,-13.739,83.889,175.8304,-0.8156,0.0000
C00632=-82.242,-12.615,80.917,179.8768,-0.0322,0.0000
C00633=-78.920,-10.667,78.774,-164.1411,19.9540,0.0000
C00634=-78.109,-6.557,77.927,-177.3739,35.8809,0.0000
C00635=-78.242,-2.973,77.891,178.0849,36.5897,0.0000
C00636=-78.293,0.000,77.915,179.9992,36.6075,0.0000
C00637=-78.242,2.972,77.891,-178.0840,36.5898,0.0000
C00638=-78.109,6.557,77.927,177.3711,35.8803,0.0000
C00639=-78.920,10.668,78.775,164.1412,19.9538,0.0000
C00640=-82.242,12.615,80.917,-179.8768,-0.0322,0.0000
C00641=-87.966,13.739,83.889,-175.8304,-0.8156,0.0000
C00642=-95.594,14.847,86.955,-174.0306,-1.0511,0.0000
C00643=-104.122,16.063,89.294,-172.8761,-1.2698,0.0000
C00644=-112.004,17.555,90.443,-173.2337,-2.5774,0.0000
C00645=-117.762,21.842,91.047,-177.2449,-3.6485,0.0000
C00646=-120.509,28.456,91.537,-179.6908,-2.2187,0.0000
C00647=-119.647,36.055,92.031,179.9584,-0.1409,0.0000
C00648=-117.032,43.902,92.356,179.9939,-0.0163,0.0000
C00649=-113.797,51.711,92.356,179.9928,-0.0158,0.0000
C00650=-110.098,59.109,92.031,179.9297,-0.1290,0.0000
C00651=-105.334,65.092,91.537,178.2123,-1.3507,0.0000
C00652=-98.715,67.825,91.047,175.4764,-0.6337,0.0000
C00653=-91.612,66.785,90.443,173.3988,2.9804,0.0000
C00654=-84.984,62.267,89.294,174.0598,4.1581,0.0000
C00655=-78.094,57.097,86.955,175.0328,3.4887,0.0000
C00656=-71.917,52.487,83.889,176.4742,2.3755,0.0000
C00657=-67.074,49.233,80.917,179.8901,0.0644,0.0000
C00658=-63.348,48.262,78.774,-155.4112,3.1965,0.0000
C00659=-59.868,50.595,77.927,-151.4568,25.5976,0.0000
C00660=-57.428,53.224,77.891,-153.3753,28.7488,0.0000
C00661=-55.362,55.362,77.915,-152.2881,27.7128,0.0000
C00662=-53.224,57.427,77.891,-151.2507,26.6243,0.0000
C00663=-50.595,59.868,77.927,-154.4045,28.5442,0.0000
C00664=-48.262,63.348,78.775,-176.8036,24.5886,0.0000
C00665=-49.233,67.074,80.917,-179.9356,-0.1099,0.0000
C00666=-52.487,71.917,83.889,-177.6245,-3.5258,0.0000
C00667=-57.097,78.094,86.955,-176.5113,-4.9672,0.0000
C00668=-62.267,84.984,89.294,-175.8419,-5.9402,0.0000
C00669=-66.785,91.612,90.443,-177.0196,-6.6012,0.0000
C00670=-67.825,98.715,91.047,179.3663,-4.5236,0.0000
C00671=-65.092,105.334,91.537,178.6493,-1.7877,0.0000
C00672=-59.109,110.098,92.031,179.8710,-0.0703,0.0000
C00673=-51.711,113.797,92.356,179.9842,-0.0072,0.0000
C00674=-43.902,117.032,92.356,179.9837,-0.0061,0.0000
C00675=-36.055,119.647,92.031,179.8591,-0.0416,0.0000
C00676=-28.456,120.509,91.537,177.7813,0.3092,0.0000
C00677=-21.842,117.762,91.047,176.3515,2.7551,0.0000
C00678=-17.555,112.004,90.443,177.4226,6.7663,0.0000
C00679=-16.063,104.122,89.294,178.7302,7.1239,0.0000
C00680=-14.847,95.594,86.955,178.9489,5.9694,0.0000
C00681=-13.739,87.966,83.889,179.1844,4.1696,0.0000
C00682=-12.615,82.242,80.917,179.9678,0.1232,0.0000
C00683=-10.668,78.920,78.775,-160.0462,-15.8588,0.0000
C00684=-6.557,78.109,77.927,-144.1197,-2.6289,0.0000
C00685=-2.972,78.242,77.891,-143.4102,1.9160,0.0000
C00686=0.000,78.293,77.915,-143.3925,-0.0008,0.0000
C00687=0.000,76.990,79.688,-143.9716,-0.0008,0.0000
C00688=2.854,76.943,79.662,-143.9881,-1.8387,0.0000
C00689=6.357,76.822,79.700,-144.7522,2.8648,0.0000
C00690=10.424,77.685,80.579,-161.2040,15.5406,0.0000
C00691=12.323,81.140,82.798,179.8614,-0.5603,0.0000
C00692=13.416,87.068,85.872,179.2048,-4.2286,0.0000
C00693=14.514,94.942,89.029,179.0062,-5.8363,0.0000
C00694=15.722,103.716,91.429,178.8210,-6.8702,0.0000
C00695=17.195,111.808,92.604,177.5896,-6.5176,0.0000
C00696=21.508,117.721,93.221,176.5147,-2.6826,0.0000
C00697=28.195,120.557,93.721,177.8730,-0.3071,0.0000
C00698=35.892,119.701,94.224,179.8645,0.0399,0.0000
C00699=43.847,117.053,94.555,179.9844,0.0058,0.0000
C00700=51.765,113.773,94.555,179.9848,0.0069,0.0000
C00701=59.262,110.021,94.224,179.8760,0.0676,0.0000
C00702=65.310,105.183,93.721,178.7126,1.7214,0.0000
C00703=68.033,98.450,93.221,179.4308,4.3574,0.0000
C00704=66.901,91.219,92.604,-177.0793,6.3084,0.0000
C00705=62.221,84.456,91.429,-175.9592,5.6963,0.0000
C00706=56.872,77.397,89.029,-176.5657,4.8325,0.0000
C00707=52.080,71.053,85.872,-177.5683,3.5532,0.0000
C00708=48.661,66.088,82.798,-179.7018,0.4942,0.0000
C00709=47.561,62.302,80.579,-177.4791,-23.6199,0.0000
C00710=49.827,58.816,79.700,-155.0942,-28.1503,0.0000
C00711=52.389,56.425,79.662,-151.7790,-26.1634,0.0000
C00712=54.440,54.440,79.688,-152.7837,-27.2153,0.0000
C00713=56.425,52.390,79.662,-153.8371,-28.2215,0.0000
C00714=58.817,49.826,79.700,-151.8487,-24.9036,0.0000
C00715=62.302,47.561,80.579,-156.3803,-2.5207,0.0000
C00716=66.088,48.661,82.798,179.5058,-0.2982,0.0000
C00717=71.053,52.080,85.872,176.4468,-2.4317,0.0000
C00718=77.397,56.872,89.029,175.1675,-3.4343,0.0000
C00719=84.456,62.221,91.429,174.3037,-4.0408,0.0000
C00720=91.219,66.901,92.604,173.6916,-2.9207,0.0000
C00721=98.450,68.033,93.221,175.6426,0.5692,0.0000
C00722=105.183,65.310,93.721,178.2786,1.2874,0.0000
C00723=110.021,59.262,94.224,179.9324,0.1240,0.0000
C00724=113.773,51.765,94.555,179.9931,0.0152,0.0000
C00725=117.053,43.847,94.555,179.9942,0.0156,0.0000
C00726=119.701,35.892,94.224,179.9601,0.1355,0.0000
C00727=120.557,28.195,93.721,-179.6929,2.1270,0.0000
C00728=117.721,21.508,93.221,-177.3174,3.4853,0.0000
C00729=111.808,17.195,92.604,-173.4824,2.4104,0.0000
C00730=103.716,15.722,91.429,-173.1298,1.1790,0.0000
C00731=94.942,14.514,89.029,-174.1637,0.9938,0.0000
C00732=87.068,13.416,85.872,-175.7714,0.7952,0.0000
C00733=81.140,12.323,82.798,-179.4397,0.1386,0.0000
C00734=77.685,10.424,80.579,164.4594,-18.7960,0.0000
C00735=76.822,6.357,79.700,177.1352,-35.2478,0.0000
C00736=76.943,2.854,79.662,-178.1613,-36.0119,0.0000
C00737=76.990,0.000,79.688,-179.9992,-36.0284,0.0000
C00738=76.943,-2.853,79.662,178.1604,-36.0119,0.0000
C00739=76.822,-6.357,79.700,-177.1324,-35.2471,0.0000
C00740=77.685,-10.424,80.579,-164.4594,-18.7957,0.0000
C00741=81.140,-12.323,82.798,179.4397,0.1386,0.0000
C00742=87.068,-13.416,85.872,175.7714,0.7952,0.0000
C00743=94.942,-14.514,89.029,174.1637,0.9938,0.0000
C00744=103.716,-15.722,91.429,173.1298,1.1790,0.0000
C00745=111.808,-17.195,92.604,173.4824,2.4104,0.0000
C00746=117.721,-21.508,93.221,177.3174,3.4853,0.0000
C00747=120.557,-28.195,93.721,179.6929,2.1270,0.0000
C00748=119.701,-35.892,94.224,-179.9601,0.1355,0.0000
C00749=117.053,-43.847,94.555,-179.9942,0.0156,0.0000
C00750=113.773,-51.765,94.555,-179.9931,0.0152,0.0000
C00751=110.021,-59.262,94.224,-179.9324,0.1240,0.0000
C00752=105.183,-65.310,93.721,-178.2786,1.2874,0.0000
C00753=98.450,-68.033,93.221,-175.6426,0.5692,0.0000
C00754=91.219,-66.901,92.604,-173.6916,-2.9207,0.0000
C00755=84.456,-62.221,91.429,-174.3037,-4.0408,0.0000
C00756=77.397,-56.872,89.029,-175.1675,-3.4343,0.0000
C00757=71.053,-52.080,85.872,-176.4468,-2.4317,0.0000
C00758=66.088,-48.661,82.798,-179.5058,-0.2982,0.0000
C00759=62.302,-47.561,80.579,156.3801,-2.5209,0.0000
C00760=58.816,-49.827,79.700,151.8497,-24.9058,0.0000
C00761=56.425,-52.389,79.662,153.8366,-28.2210,0.0000
C00762=54.440,-54.440,79.688,152.7847,-27.2163,0.0000
C00763=52.390,-56.425,79.662,151.7785,-26.1629,0.0000
C00764=49.826,-58.817,79.700,155.0964,-28.1513,0.0000
C00765=47.561,-62.302,80.579,177.4793,-23.6197,0.0000
C00766=48.661,-66.088,82.798,179.7018,0.4942,0.0000
C00767=52.080,-71.053,85.872,177.5683,3.5532,0.0000
C00768=56.872,-77.397,89.029,176.5657,4.8325,0.0000
C00769=62.221,-84.456,91.429,175.9592,5.6963,0.0000
C00770=66.901,-91.219,92.604,177.0793,6.3084,0.0000
C00771=68.033,-98.450,93.221,-179.4308,4.3574,0.0000
C00772=65.310,-105.183,93.721,-178.7126,1.7214,0.0000
C00773=59.262,-110.021,94.224,-179.8760,0.0676,0.0000
C00774=51.765,-113.773,94.555,-179.9848,0.0069,0.0000
C00775=43.847,-117.053,94.555,-179.9844,0.0058,0.0000
C00776=35.892,-119.701,94.224,-179.8645,0.0399,0.0000
C00777=28.195,-120.557,93.721,-177.8730,-0.3071,0.0000
C00778=21.508,-117.721,93.221,-176.5147,-2.6826,0.0000
C00779=17.195,-111.808,92.604,-177.5896,-6.5176,0.0000
C00780=15.722,-103.716,91.429,-178.8210,-6.8702,0.0000
C00781=14.514,-94.942,89.029,-179.0062,-5.8363,0.0000
C00782=13.416,-87.068,85.872,-179.2048,-4.2286,0.0000
C00783=12.323,-81.140,82.798,-179.8614,-0.5603,0.0000
C00784=10.424,-77.685,80.579,161.2040,15.5406,0.0000
C00785=6.357,-76.822,79.700,144.7522,2.8648,0.0000
C00786=2.854,-76.943,79.662,143.9881,-1.8387,0.0000
C00787=0.000,-76.990,79.688,143.9716,-0.0008,0.0000
C00788=0.000,-76.990,79.688,143.9716,-0.0008,0.0000
C00789=-2.853,-76.943,79.662,143.9881,1.8396,0.0000
C00790=-6.357,-76.822,79.700,144.7529,-2.8676,0.0000
C00791=-10.424,-77.685,80.579,161.2043,-15.5406,0.0000
C00792=-12.323,-81.140,82.798,-179.8614,0.5603,0.0000
C00793=-13.416,-87.068,85.872,-179.2048,4.2286,0.0000
C00794=-14.514,-94.942,89.029,-179.0062,5.8363,0.0000
C00795=-15.722,-103.716,91.429,-178.8210,6.8702,0.0000
C00796=-17.195,-111.808,92.604,-177.5896,6.5176,0.0000
C00797=-21.508,-117.721,93.221,-176.5147,2.6826,0.0000
C00798=-28.195,-120.557,93.721,-177.8730,0.3071,0.0000
C00799=-35.892,-119.701,94.224,-179.8645,-0.0399,0.0000
C00800=-43.847,-117.053,94.555,-179.9844,-0.0058,0.0000
C00801=-51.765,-113.773,94.555,-179.9848,-0.0069,0.0000
C00802=-59.262,-110.021,94.224,-179.8760,-0.0676,0.0000
C00803=-65.310,-105.183,93.721,-178.7126,-1.7214,0.0000
C00804=-68.033,-98.450,93.221,-179.4308,-4.3574,0.0000
C00805=-66.901,-91.219,92.604,177.0793,-6.3084,0.0000
C00806=-62.221,-84.456,91.429,175.9592,-5.6963,0.0000
C00807=-56.872,-77.397,89.029,176.5657,-4.8325,0.0000
C00808=-52.080,-71.053,85.872,177.5683,-3.5532,0.0000
C00809=-48.661,-66.088,82.798,179.7018,-0.4942,0.0000
C00810=-47.561,-62.302,80.579,177.4791,23.6199,0.0000
C00811=-49.827,-58.816,79.700,155.0942,28.1503,0.0000
C00812=-52.389,-56.425,79.662,151.7790,26.1634,0.0000
C00813=-54.440,-54.440,79.688,152.7837,27.2153,0.0000
C00814=-56.425,-52.390,79.662,153.8371,28.2215,0.0000
C00815=-58.817,-49.826,79.700,151.8487,24.9036,0.0000
C00816=-62.302,-47.561,80.579,156.3803,2.5207,0.0000
C00817=-66.088,-48.661,82.798,-179.5058,0.2982,0.0000
C00818=-71.053,-52.080,85.872,-176.4468,2.4317,0.0000
C00819=-77.397,-56.872,89.029,-175.1675,3.4343,0.0000
C00820=-84.456,-62.221,91.429,-174.3037,4.0408,0.0000
C00821=-91.219,-66.901,92.604,-173.6916,2.9207,0.0000
C00822=-98.450,-68.033,93.221,-175.6426,-0.5692,0.0000
C00823=-105.183,-65.310,93.721,-178.2786,-1.2874,0.0000
C00824=-110.021,-59.262,94.224,-179.9324,-0.1240,0.0000
C00825=-113.773,-51.765,94.555,-179.9931,-0.0152,0.0000
C00826=-117.053,-43.847,94.555,-179.9942,-0.0156,0.0000
C00827=-119.701,-35.892,94.224,-179.9601,-0.1355,0.0000
C00828=-120.557,-28.195,93.721,179.6929,-2.1270,0.0000
C00829=-117.721,-21.508,93.221,177.3174,-3.4853,0.0000
C00830=-111.808,-17.195,92.604,173.4824,-2.4104,0.0000
C00831=-103.716,-15.722,91.429,173.1298,-1.1790,0.0000
C00832=-94.942,-14.514,89.029,174.1637,-0.9938,0.0000
C00833=-87.068,-13.416,85.872,175.7714,-0.7952,0.0000
C00834=-81.140,-12.323,82.798,179.4397,-0.1386,0.0000
C00835=-77.685,-10.424,80.579,-164.4594,18.7960,0.0000
C00836=-76.822,-6.357,79.700,-177.1352,35.2478,0.0000
C00837=-76.943,-2.854,79.662,178.1613,36.0119,0.0000
C00838=-76.990,0.000,79.688,179.9992,36.0284,0.0000
C00839=-76.943,2.853,79.662,-178.1604,36.0119,0.0000
C00840=-76.822,6.357,79.700,177.1324,35.2471,0.0000
C00841=-77.685,10.424,80.579,164.4594,18.7957,0.0000
C00842=-81.140,12.323,82.798,-179.4397,-0.1386,0.0000
C00843=-87.068,13.416,85.872,-175.7714,-0.7952,0.0000
C00844=-94.942,14.514,89.029,-174.1637,-0.9938,0.0000
C00845=-103.716,15.722,91.429,-173.1298,-1.1790,0.0000
C00846=-111.808,17.195,92.604,-173.4824,-2.4104,0.0000
C00847=-117.721,21.508,93.221,-177.3174,-3.4853,0.0000
C00848=-120.557,28.195,93.721,-179.6929,-2.1270,0.0000
C00849=-119.701,35.892,94.224,179.9601,-0.1355,0.0000
C00850=-117.053,43.847,94.555,179.9942,-0.0156,0.0000
C00851=-113.773,51.765,94.555,179.9931,-0.0152,0.0000
C00852=-110.021,59.262,94.224,179.9324,-0.1240,0.0000
C00853=-105.183,65.310,93.721,178.2786,-1.2874,0.0000
C00854=-98.450,68.033,93.221,175.6426,-0.5692,0.0000
C00855=-91.219,66.901,92.604,173.6916,2.9207,0.0000
C00856=-84.456,62.221,91.429,174.3037,4.0408,0.0000
C00857=-77.397,56.872,89.029,175.1675,3.4343,0.0000
C00858=-71.053,52.080,85.872,176.4468,2.4317,0.0000
C00859=-66.088,48.661,82.798,179.5058,0.2982,0.0000
C00860=-62.302,47.561,80.579,-156.3801,2.5209,0.0000
C00861=-58.816,49.827,79.700,-151.8497,24.9058,0.0000
C00862=-56.425,52.389,79.662,-153.8366,28.2210,0.0000
C00863=-54.440,54.440,79.688,-152.7847,27.2163,0.0000
C00864=-52.390,56.425,79.662,-151.7785,26.1629,0.0000
C00865=-49.826,58.817,79.700,-155.0964,28.1513,0.0000
C00866=-47.561,62.302,80.579,-177.4793,23.6197,0.0000
C00867=-48.661,66.088,82.798,-179.7018,-0.4942,0.0000
C00868=-52.080,71.053,85.872,-177.5683,-3.5532,0.0000
C00869=-56.872,77.397,89.029,-176.5657,-4.8325,0.0000
C00870=-62.221,84.456,91.429,-175.9592,-5.6963,0.0000
C00871=-66.901,91.219,92.604,-177.0793,-6.3084,0.0000
C00872=-68.033,98.450,93.221,179.4308,-4.3574,0.0000
C00873=-65.310,105.183,93.721,178.7126,-1.7214,0.0000
C00874=-59.262,110.021,94.224,179.8760,-0.0676,0.0000
C00875=-51.765,113.773,94.555,179.9848,-0.0069,0.0000
C00876=-43.847,117.053,94.555,179.9844,-0.0058,0.0000
C00877=-35.892,119.701,94.224,179.8645,-0.0399,0.0000
C00878=-28.195,120.557,93.721,177.8730,0.3071,0.0000
C00879=-21.508,117.721,93.221,176.5147,2.6826,0.0000
C00880=-17.195,111.808,92.604,177.5896,6.5176,0.0000
C00881=-15.722,103.716,91.429,178.8210,6.8702,0.0000
C00882=-14.514,94.942,89.029,179.0062,5.8363,0.0000
C00883=-13.416,87.068,85.872,179.2048,4.2286,0.0000
C00884=-12.323,81.140,82.798,179.8614,0.5603,0.0000
C00885=-10.424,77.685,80.579,-161.2043,-15.5406,0.0000
C00886=-6.357,76.822,79.700,-144.7529,-2.8676,0.0000
C00887=-2.853,76.943,79.662,-143.9881,1.8396,0.0000
C00888=0.000,76.990,79.688,-143.9716,-0.0008,0.0000
C00889=0.000,75.706,81.474,-144.6196,-0.0009,0.0000
C00890=2.736,75.663,81.448,-144.6347,-1.7577,0.0000
C00891=6.159,75.554,81.487,-145.4561,3.0860,0.0000
C00892=10.184,76.470,82.397,-162.3577,15.1555,0.0000
C00893=12.037,80.061,84.694,179.7790,-0.9434,0.0000
C00894=13.103,86.196,87.867,179.2309,-4.2469,0.0000
C00895=14.193,94.316,91.114,179.0654,-5.6654,0.0000
C00896=15.398,103.330,93.571,178.9112,-6.5757,0.0000
C00897=16.854,111.622,94.770,177.7603,-6.2249,0.0000
C00898=21.193,117.683,95.398,176.6983,-2.5860,0.0000
C00899=27.948,120.602,95.907,177.9788,-0.3012,0.0000
C00900=35.739,119.751,96.419,179.8710,0.0379,0.0000
C00901=43.796,117.073,96.755,179.9852,0.0055,0.0000
C00902=51.815,113.751,96.755,179.9856,0.0066,0.0000
C00903=59.406,109.948,96.419,179.8820,0.0644,0.0000
C00904=65.516,105.041,95.907,178.7834,1.6423,0.0000
C00905=68.229,98.200,95.398,179.4926,4.1597,0.0000
C00906=67.011,90.846,94.770,-177.1678,5.9818,0.0000
C00907=62.177,83.953,93.571,-176.1058,5.4240,0.0000
C00908=56.655,76.728,91.114,-176.6456,4.6697,0.0000
C00909=51.685,70.215,87.867,-177.5369,3.5478,0.0000
C00910=48.100,65.123,84.694,-179.4892,0.8234,0.0000
C00911=46.871,61.274,82.397,-178.0896,-22.6073,0.0000
C00912=49.069,57.780,81.487,-155.8363,-27.6951,0.0000
C00913=51.567,55.437,81.448,-152.3648,-25.6489,0.0000
C00914=53.532,53.532,81.474,-153.3359,-26.6631,0.0000
C00915=55.437,51.568,81.448,-154.3516,-27.6357,0.0000
C00916=57.780,49.069,81.487,-152.3039,-24.1615,0.0000
C00917=61.274,46.871,82.397,-157.3930,-1.9101,0.0000
C00918=65.123,48.100,84.694,179.1766,-0.5108,0.0000
C00919=70.215,51.685,87.867,176.4522,-2.4631,0.0000
C00920=76.728,56.655,91.114,175.3303,-3.3544,0.0000
C00921=83.953,62.177,93.571,174.5760,-3.8942,0.0000
C00922=90.846,67.011,94.770,174.0182,-2.8322,0.0000
C00923=98.200,68.229,95.398,175.8403,0.5074,0.0000
C00924=105.041,65.516,95.907,178.3577,1.2166,0.0000
C00925=109.948,59.406,96.419,179.9356,0.1180,0.0000
C00926=113.751,51.815,96.755,179.9934,0.0144,0.0000
C00927=117.073,43.796,96.755,179.9945,0.0148,0.0000
C00928=119.751,35.739,96.419,179.9621,0.1290,0.0000
C00929=120.602,27.948,95.907,-179.6988,2.0212,0.0000
C00930=117.683,21.193,95.398,-177.4140,3.3017,0.0000
C00931=111.622,16.854,94.770,-173.7751,2.2397,0.0000
C00932=103.330,15.398,93.571,-173.4243,1.0888,0.0000
C00933=94.316,14.193,91.114,-174.3346,0.9346,0.0000
C00934=86.196,13.103,87.867,-175.7531,0.7691,0.0000
C00935=80.061,12.037,84.694,-179.0566,0.2210,0.0000
C00936=76.470,10.184,82.397,164.8445,-17.6423,0.0000
C00937=75.554,6.159,81.487,176.9140,-34.5439,0.0000
C00938=75.663,2.736,81.448,-178.2423,-35.3653,0.0000
C00939=75.706,0.000,81.474,-179.9991,-35.3804,0.0000
C00940=75.663,-2.736,81.448,178.2414,-35.3653,0.0000
C00941=75.554,-6.160,81.487,-176.9112,-34.5432,0.0000
C00942=76.470,-10.184,82.397,-164.8445,-17.6419,0.0000
C00943=80.061,-12.037,84.694,179.0566,0.2210,0.0000
C00944=86.196,-13.103,87.867,175.7531,0.7691,0.0000
C00945=94.316,-14.193,91.114,174.3346,0.9346,0.0000
C00946=103.330,-15.398,93.571,173.4243,1.0888,0.0000
C00947=111.622,-16.854,94.770,173.7751,2.2397,0.0000
C00948=117.683,-21.193,95.398,177.4140,3.3017,0.0000
C00949=120.602,-27.948,95.907,179.6988,2.0212,0.0000
C00950=119.751,-35.739,96.419,-179.9621,0.1290,0.0000
C00951=117.073,-43.796,96.755,-179.9945,0.0148,0.0000
C00952=113.751,-51.815,96.755,-179.9934,0.0144,0.0000
C00953=109.948,-59.406,96.419,-179.9356,0.1180,0.0000
C00954=105.041,-65.516,95.907,-178.3577,1.2166,0.0000
C00955=98.200,-68.229,95.398,-175.8403,0.5074,0.0000
C00956=90.846,-67.011,94.770,-174.0182,-2.8322,0.0000
C00957=83.953,-62.177,93.571,-174.5760,-3.8942,0.0000
C00958=76.728,-56.655,91.114,-175.3303,-3.3544,0.0000
C00959=70.215,-51.685,87.867,-176.4522,-2.4631,0.0000
C00960=65.123,-48.100,84.694,-179.1766,-0.5108,0.0000
C00961=61.274,-46.871,82.397,157.3927,-1.9104,0.0000
C00962=57.780,-49.069,81.487,152.3049,-24.1637,0.0000
C00963=55.437,-51.567,81.448,154.3511,-27.6352,0.0000
C00964=53.532,-53.532,81.474,153.3369,-26.6641,0.0000
C00965=51.568,-55.437,81.448,152.3643,-25.6484,0.0000
C00966=49.069,-57.780,81.487,155.8385,-27.6961,0.0000
C00967=46.871,-61.274,82.397,178.0899,-22.6070,0.0000
C00968=48.100,-65.123,84.694,179.4892,0.8234,0.0000
C00969=51.685,-70.215,87.867,177.5369,3.5478,0.0000
C00970=56.655,-76.728,91.114,176.6456,4.6697,0.0000
C00971=62.177,-83.953,93.571,176.1058,5.4240,0.0000
C00972=67.011,-90.846,94.770,177.1678,5.9818,0.0000
C00973=68.229,-98.200,95.398,-179.4926,4.1597,0.0000
C00974=65.516,-105.041,95.907,-178.7834,1.6423,0.0000
C00975=59.406,-109.948,96.419,-179.8820,0.0644,0.0000
C00976=51.815,-113.751,96.755,-179.9856,0.0066,0.0000
C00977=43.796,-117.073,96.755,-179.9852,0.0055,0.0000
C00978=35.739,-119.751,96.419,-179.8710,0.0379,0.0000
C00979=27.948,-120.602,95.907,-177.9788,-0.3012,0.0000
C00980=21.193,-117.683,95.398,-176.6983,-2.5860,0.0000
C00981=16.854,-111.622,94.770,-177.7603,-6.2249,0.0000
C00982=15.398,-103.330,93.571,-178.9112,-6.5757,0.0000
C00983=14.193,-94.316,91.114,-179.0654,-5.6654,0.0000
C00984=13.103,-86.196,87.867,-179.2309,-4.2469,0.0000
C00985=12.037,-80.061,84.694,-179.7790,-0.9434,0.0000
C00986=10.184,-76.470,82.397,162.3577,15.1555,0.0000
C00987=6.159,-75.554,81.487,145.4561,3.0860,0.0000
C00988=2.736,-75.663,81.448,144.6347,-1.7577,0.0000
C00989=0.000,-75.706,81.474,144.6196,-0.0009,0.0000
C00990=0.000,-75.706,81.474,144.6196,-0.0009,0.0000
C00991=-2.736,-75.663,81.448,144.6347,1.7586,0.0000
C00992=-6.160,-75.554,81.487,145.4568,-3.0888,0.0000
C00993=-10.184,-76.470,82.397,162.3581,-15.1555,0.0000
C00994=-12.037,-80.061,84.694,-179.7790,0.9434,0.0000
C00995=-13.103,-86.196,87.867,-179.2309,4.2469,0.0000
C00996=-14.193,-94.316,91.114,-179.0654,5.6654,0.0000
C00997=-15.398,-103.330,93.571,-178.9112,6.5757,0.0000
C00998=-16.854,-111.622,94.770,-177.7603,6.2249,0.0000
C00999=-21.193,-117.683,95.398,-176.6983,2.5860,0.0000
C01000=-27.948,-120.602,95.907,-177.9788,0.3012,0.0000
C01001=-35.739,-119.751,96.419,-179.8710,-0.0379,0.0000
C01002=-43.796,-117.073,96.755,-179.9852,-0.0055,0.0000
C01003=-51.815,-113.751,96.755,-179.9856,-0.0066,0.0000
C01004=-59.406,-109.948,96.419,-179.8820,-0.0644,0.0000
C01005=-65.516,-105.041,95.907,-178.7834,-1.6423,0.0000
C01006=-68.229,-98.200,95.398,-179.4926,-4.1597,0.0000
C01007=-67.011,-90.846,94.770,177.1678,-5.9818,0.0000
C01008=-62.177,-83.953,93.571,176.1058,-5.4240,0.0000
C01009=-56.655,-76.728,91.114,176.6456,-4.6697,0.0000
C01010=-51.685,-70.215,87.867,177.5369,-3.5478,0.0000
C01011=-48.100,-65.123,84.694,179.4892,-0.8234,0.0000
C01012=-46.871,-61.274,82.397,178.0896,22.6073,0.0000
C01013=-49.069,-57.780,81.487,155.8363,27.6951,0.0000
C01014=-51.567,-55.437,81.448,152.3648,25.6489,0.0000
C01015=-53.532,-53.532,81.474,153.3359,26.6631,0.0000
C01016=-55.437,-51.568,81.448,154.3516,27.6357,0.0000
C01017=-57.780,-49.069,81.487,152.3039,24.1615,0.0000
C01018=-61.274,-46.871,82.397,157.3930,1.9101,0.0000
C01019=-65.123,-48.100,84.694,-179.1766,0.5108,0.0000
C01020=-70.215,-51.685,87.867,-176.4522,2.4631,0.0000
C01021=-76.728,-56.655,91.114,-175.3303,3.3544,0.0000
C01022=-83.953,-62.177,93.571,-174.5760,3.8942,0.0000
C01023=-90.846,-67.011,94.770,-174.0182,2.8322,0.0000
C01024=-98.200,-68.229,95.398,-175.8403,-0.5074,0.0000
C01025=-105.041,-65.516,95.907,-178.3577,-1.2166,0.0000
C01026=-109.948,-59.406,96.419,-179.9356,-0.1180,0.0000
C01027=-113.751,-51.815,96.755,-179.9934,-0.0144,0.0000
C01028=-117.073,-43.796,96.755,-179.9945,-0.0148,0.0000
C01029=-119.751,-35.739,96.419,-179.9621,-0.1290,0.0000
C01030=-120.602,-27.948,95.907,179.6988,-2.0212,0.0000
C01031=-117.683,-21.193,95.398,177.4140,-3.3017,0.0000
C01032=-111.622,-16.854,94.770,173.7751,-2.2397,0.0000
C01033=-103.330,-15.398,93.571,173.4243,-1.0888,0.0000
C01034=-94.316,-14.193,91.114,174.3346,-0.9346,0.0000
C01035=-86.196,-13.103,87.867,175.7531,-0.7691,0.0000
C01036=-80.061,-12.037,84.694,179.0566,-0.2210,0.0000
C01037=-76.470,-10.184,82.397,-164.8445,17.6423,0.0000
C01038=-75.554,-6.159,81.487,-176.9140,34.5439,0.0000
C01039=-75.663,-2.736,81.448,178.2423,35.3653,0.0000
C01040=-75.706,0.000,81.474,179.9991,35.3804,0.0000
C01041=-75.663,2.736,81.448,-178.2414,35.3653,0.0000
C01042=-75.554,6.160,81.487,176.9112,34.5432,0.0000
C01043=-76.470,10.184,82.397,164.8445,17.6419,0.0000
C01044=-80.061,12.037,84.694,-179.0566,-0.2210,0.0000
C01045=-86.196,13.103,87.867,-175.7531,-0.7691,0.0000
C01046=-94.316,14.193,91.114,-174.3346,-0.9346,0.0000
C01047=-103.330,15.398,93.571,-173.4243,-1.0888,0.0000
C01048=-111.622,16.854,94.770,-173.7751,-2.2397,0.0000
C01049=-117.683,21.193,95.398,-177.4140,-3.3017,0.0000
C01050=-120.602,27.948,95.907,-179.6988,-2.0212,0.0000
C01051=-119.751,35.739,96.419,179.9621,-0.1290,0.0000
C01052=-117.073,43.796,96.755,179.9945,-0.0148,0.0000
C01053=-113.751,51.815,96.755,179.9934,-0.0144,0.0000
C01054=-109.948,59.406,96.419,179.9356,-0.1180,0.0000
C01055=-105.041,65.516,95.907,178.3577,-1.2166,0.0000
C01056=-98.200,68.229,95.398,175.8403,-0.5074,0.0000
C01057=-90.846,67.011,94.770,174.0182,2.8322,0.0000
C01058=-83.953,62.177,93.571,174.5760,3.8942,0.0000
C01059=-76.728,56.655,91.114,175.3303,3.3544,0.0000
C01060=-70.215,51.685,87.867,176.4522,2.4631,0.0000
C01061=-65.123,48.100,84.694,179.1766,0.5108,0.0000
C01062=-61.274,46.871,82.397,-157.3927,1.9104,0.0000
C01063=-57.780,49.069,81.487,-152.3049,24.1637,0.0000
C01064=-55.437,51.567,81.448,-154.3511,27.6352,0.0000
C01065=-53.532,53.532,81.474,-153.3369,26.6641,0.0000
C01066=-51.568,55.437,81.448,-152.3643,25.6484,0.0000
C01067=-49.069,57.780,81.487,-155.8385,27.6961,0.0000
C01068=-46.871,61.274,82.397,-178.0899,22.6070,0.0000
C01069=-48.100,65.123,84.694,-179.4892,-0.8234,0.0000
C01070=-51.685,70.215,87.867,-177.5369,-3.5478,0.0000
C01071=-56.655,76.728,91.114,-176.6456,-4.6697,0.0000
C01072=-62.177,83.953,93.571,-176.1058,-5.4240,0.0000
C01073=-67.011,90.846,94.770,-177.1678,-5.9818,0.0000
C01074=-68.229,98.200,95.398,179.4926,-4.1597,0.0000
C01075=-65.516,105.041,95.907,178.7834,-1.6423,0.0000
C01076=-59.406,109.948,96.419,179.8820,-0.0644,0.0000
C01077=-51.815,113.751,96.755,179.9856,-0.0066,0.0000
C01078=-43.796,117.073,96.755,179.9852,-0.0055,0.0000
C01079=-35.739,119.751,96.419,179.8710,-0.0379,0.0000
C01080=-27.948,120.602,95.907,177.9788,0.3012,0.0000
C01081=-21.193,117.683,95.398,176.6983,2.5860,0.0000
C01082=-16.854,111.622,94.770,177.7603,6.2249,0.0000
C01083=-15.398,103.330,93.571,178.9112,6.5757,0.0000
C01084=-14.193,94.316,91.114,179.0654,5.6654,0.0000
C01085=-13.103,86.196,87.867,179.2309,4.2469,0.0000
C01086=-12.037,80.061,84.694,179.7790,0.9434,0.0000
C01087=-10.184,76.470,82.397,-162.3581,-15.1555,0.0000
C01088=-6.160,75.554,81.487,-145.4568,-3.0888,0.0000
C01089=-2.736,75.663,81.448,-144.6347,1.7586,0.0000
C01090=0.000,75.706,81.474,-144.6196,-0.0009,0.0000
C01091=0.000,74.443,83.276,-145.3411,-0.0009,0.0000
C01092=2.621,74.405,83.248,-145.3548,-1.6723,0.0000
C01093=5.965,74.307,83.289,-146.2348,3.2868,0.0000
C01094=9.949,75.277,84.231,-163.5015,14.7075,0.0000
C01095=11.757,79.007,86.605,179.7171,-1.2728,0.0000
C01096=12.799,85.352,89.876,179.2620,-4.2251,0.0000
C01097=13.887,93.717,93.208,179.1263,-5.4571,0.0000
C01098=15.091,102.965,95.718,179.0007,-6.2410,0.0000
C01099=16.532,111.447,96.939,177.9343,-5.8891,0.0000
C01100=20.897,117.648,97.578,176.9018,-2.4653,0.0000
C01101=27.718,120.644,98.094,178.0988,-0.2913,0.0000
C01102=35.596,119.798,98.613,179.8785,0.0356,0.0000
C01103=43.748,117.091,98.954,179.9861,0.0052,0.0000
C01104=51.862,113.730,98.954,179.9865,0.0062,0.0000
C01105=59.540,109.881,98.613,179.8889,0.0607,0.0000
C01106=65.708,104.908,98.094,178.8613,1.5505,0.0000
C01107=68.413,97.966,97.578,179.5514,3.9310,0.0000
C01108=67.115,90.495,96.939,-177.2844,5.6222,0.0000
C01109=62.136,83.478,95.718,-176.2813,5.1236,0.0000
C01110=56.449,76.088,93.208,-176.7508,4.4792,0.0000
C01111=51.303,69.404,89.876,-177.5304,3.5105,0.0000
C01112=47.553,64.180,86.605,-179.2999,1.1001,0.0000
C01113=46.194,60.264,84.231,-178.6349,-21.5560,0.0000
C01114=48.325,56.761,83.289,-156.6290,-27.1739,0.0000
C01115=50.759,54.465,83.248,-153.0117,-25.0786,0.0000
C01116=52.639,52.639,83.276,-153.9467,-26.0523,0.0000
C01117=54.465,50.759,83.248,-154.9219,-26.9888,0.0000
C01118=56.761,48.325,83.289,-152.8252,-23.3687,0.0000
C01119=60.265,46.194,84.231,-158.4444,-1.3648,0.0000
C01120=64.180,47.553,86.605,178.8999,-0.7001,0.0000
C01121=69.404,51.303,89.876,176.4895,-2.4696,0.0000
C01122=76.088,56.449,93.208,175.5208,-3.2492,0.0000
C01123=83.478,62.136,95.718,174.8764,-3.7187,0.0000
C01124=90.495,67.115,96.939,174.3778,-2.7156,0.0000
C01125=97.966,68.413,97.578,176.0690,0.4486,0.0000
C01126=104.908,65.708,98.094,178.4495,1.1387,0.0000
C01127=109.881,59.540,98.613,179.9393,0.1111,0.0000
C01128=113.730,51.862,98.954,179.9938,0.0135,0.0000
C01129=117.091,43.748,98.954,179.9948,0.0139,0.0000
C01130=119.798,35.596,98.613,179.9644,0.1215,0.0000
C01131=120.644,27.718,98.094,-179.7087,1.9012,0.0000
C01132=117.648,20.897,97.578,-177.5347,3.0982,0.0000
C01133=111.447,16.532,96.939,-174.1109,2.0657,0.0000
C01134=102.965,15.091,95.718,-173.7590,0.9993,0.0000
C01135=93.717,13.887,93.208,-174.5429,0.8737,0.0000
C01136=85.352,12.799,89.876,-175.7749,0.7380,0.0000
C01137=79.007,11.757,86.605,-178.7272,0.2829,0.0000
C01138=75.277,9.949,84.231,165.2925,-16.4985,0.0000
C01139=74.307,5.965,83.289,176.7132,-33.7652,0.0000
C01140=74.405,2.621,83.248,-178.3277,-34.6452,0.0000
C01141=74.443,0.000,83.276,-179.9991,-34.6589,0.0000
C01142=74.405,-2.620,83.248,178.3267,-34.6452,0.0000
C01143=74.307,-5.966,83.289,-176.7104,-33.7645,0.0000
C01144=75.278,-9.949,84.231,-165.2926,-16.4981,0.0000
C01145=79.007,-11.757,86.605,178.7272,0.2829,0.0000
C01146=85.352,-12.799,89.876,175.7749,0.7380,0.0000
C01147=93.717,-13.887,93.208,174.5429,0.8737,0.0000
C01148=102.965,-15.091,95.718,173.7590,0.9993,0.0000
C01149=111.447,-16.532,96.939,174.1109,2.0657,0.0000
C01150=117.648,-20.897,97.578,177.5347,3.0982,0.0000
C01151=120.644,-27.718,98.094,179.7087,1.9012,0.0000
C01152=119.798,-35.596,98.613,-179.9644,0.1215,0.0000
C01153=117.091,-43.748,98.954,-179.9948,0.0139,0.0000
C01154=113.730,-51.862,98.954,-179.9938,0.0135,0.0000
C01155=109.881,-59.540,98.613,-179.9393,0.1111,0.0000
C01156=104.908,-65.708,98.094,-178.4495,1.1387,0.0000
C01157=97.966,-68.413,97.578,-176.0690,0.4486,0.0000
C01158=90.495,-67.115,96.939,-174.3778,-2.7156,0.0000
C01159=83.478,-62.136,95.718,-174.8764,-3.7187,0.0000
C01160=76.088,-56.449,93.208,-175.5208,-3.2492,0.0000
C01161=69.404,-51.303,89.876,-176.4895,-2.4696,0.0000
C01162=64.180,-47.553,86.605,-178.8999,-0.7001,0.0000
C01163=60.264,-46.194,84.231,158.4440,-1.3651,0.0000
C01164=56.761,-48.325,83.289,152.8261,-23.3710,0.0000
C01165=54.465,-50.759,83.248,154.9214,-26.9883,0.0000
C01166=52.639,-52.639,83.276,153.9477,-26.0533,0.0000
C01167=50.759,-54.465,83.248,153.0112,-25.0781,0.0000
C01168=48.325,-56.761,83.289,156.6313,-27.1748,0.0000
C01169=46.194,-60.265,84.231,178.6352,-21.5556,0.0000
C01170=47.553,-64.180,86.605,179.2999,1.1001,0.0000
C01171=51.303,-69.404,89.876,177.5304,3.5105,0.0000
C01172=56.449,-76.088,93.208,176.7508,4.4792,0.0000
C01173=62.136,-83.478,95.718,176.2813,5.1236,0.0000
C01174=67.115,-90.495,96.939,177.2844,5.6222,0.0000
C01175=68.413,-97.966,97.578,-179.5514,3.9310,0.0000
C01176=65.708,-104.908,98.094,-178.8613,1.5505,0.0000
C01177=59.540,-109.881,98.613,-179.8889,0.0607,0.0000
C01178=51.862,-113.730,98.954,-179.9865,0.0062,0.0000
C01179=43.748,-117.091,98.954,-179.9861,0.0052,0.0000
C01180=35.596,-119.798,98.613,-179.8785,0.0356,0.0000
C01181=27.718,-120.644,98.094,-178.0988,-0.2913,0.0000
C01182=20.897,-117.648,97.578,-176.9018,-2.4653,0.0000
C01183=16.532,-111.447,96.939,-177.9343,-5.8891,0.0000
C01184=15.091,-102.965,95.718,-179.0007,-6.2410,0.0000
C01185=13.887,-93.717,93.208,-179.1263,-5.4571,0.0000
C01186=12.799,-85.352,89.876,-179.2620,-4.2251,0.0000
C01187=11.757,-79.007,86.605,-179.7171,-1.2728,0.0000
C01188=9.949,-75.277,84.231,163.5015,14.7075,0.0000
C01189=5.965,-74.307,83.289,146.2348,3.2868,0.0000
C01190=2.621,-74.405,83.248,145.3548,-1.6723,0.0000
C01191=0.000,-74.443,83.276,145.3411,-0.0009,0.0000
C01192=0.000,-74.443,83.276,145.3411,-0.0009,0.0000
C01193=-2.620,-74.405,83.248,145.3548,1.6733,0.0000
C01194=-5.966,-74.307,83.289,146.2355,-3.2896,0.0000
C01195=-9.949,-75.278,84.231,163.5019,-14.7074,0.0000
C01196=-11.757,-79.007,86.605,-179.7171,1.2728,0.0000
C01197=-12.799,-85.352,89.876,-179.2620,4.2251,0.0000
C01198=-13.887,-93.717,93.208,-179.1263,5.4571,0.0000
C01199=-15.091,-102.965,95.718,-179.0007,6.2410,0.0000
C01200=-16.532,-111.447,96.939,-177.9343,5.8891,0.0000
C01201=-20.897,-117.648,97.578,-176.9018,2.4653,0.0000
C01202=-27.718,-120.644,98.094,-178.0988,0.2913,0.0000
C01203=-35.596,-119.798,98.613,-179.8785,-0.0356,0.0000
C01204=-43.748,-117.091,98.954,-179.9861,-0.0052,0.0000
C01205=-51.862,-113.730,98.954,-179.9865,-0.0062,0.0000
C01206=-59.540,-109.881,98.613,-179.8889,-0.0607,0.0000
C01207=-65.708,-104.908,98.094,-178.8613,-1.5505,0.0000
C01208=-68.413,-97.966,97.578,-179.5514,-3.9310,0.0000
C01209=-67.115,-90.495,96.939,177.2844,-5.6222,0.0000
C01210=-62.136,-83.478,95.718,176.2813,-5.1236,0.0000
C01211=-56.449,-76.088,93.208,176.7508,-4.4792,0.0000
C01212=-51.303,-69.404,89.876,177.5304,-3.5105,0.0000
C01213=-47.553,-64.180,86.605,179.2999,-1.1001,0.0000
C01214=-46.194,-60.264,84.231,178.6349,21.5560,0.0000
C01215=-48.325,-56.761,83.289,156.6290,27.1739,0.0000
C01216=-50.759,-54.465,83.248,153.0117,25.0786,0.0000
C01217=-52.639,-52.639,83.276,153.9467,26.0523,0.0000
C01218=-54.465,-50.759,83.248,154.9219,26.9888,0.0000
C01219=-56.761,-48.325,83.289,152.8252,23.3687,0.0000
C01220=-60.265,-46.194,84.231,158.4444,1.3648,0.0000
C01221=-64.180,-47.553,86.605,-178.8999,0.7001,0.0000
C01222=-69.404,-51.303,89.876,-176.4895,2.4696,0.0000
C01223=-76.088,-56.449,93.208,-175.5208,3.2492,0.0000
C01224=-83.478,-62.136,95.718,-174.8764,3.7187,0.0000
C01225=-90.495,-67.115,96.939,-174.3778,2.7156,0.0000
C01226=-97.966,-68.413,97.578,-176.0690,-0.4486,0.0000
C01227=-104.908,-65.708,98.094,-178.4495,-1.1387,0.0000
C01228=-109.881,-59.540,98.613,-179.9393,-0.1111,0.0000
C01229=-113.730,-51.862,98.954,-179.9938,-0.0135,0.0000
C01230=-117.091,-43.748,98.954,-179.9948,-0.0139,0.0000
C01231=-119.798,-35.596,98.613,-179.9644,-0.1215,0.0000
C01232=-120.644,-27.718,98.094,179.7087,-1.9012,0.0000
C01233=-117.648,-20.897,97.578,177.5347,-3.0982,0.0000
C01234=-111.447,-16.532,96.939,174.1109,-2.0657,0.0000
C01235=-102.965,-15.091,95.718,173.7590,-0.9993,0.0000
C01236=-93.717,-13.887,93.208,174.5429,-0.8737,0.0000
C01237=-85.352,-12.799,89.876,175.7749,-0.7380,0.0000
C01238=-79.007,-11.757,86.605,178.7272,-0.2829,0.0000
C01239=-75.277,-9.949,84.231,-165.2925,16.4985,0.0000
C01240=-74.307,-5.965,83.289,-176.7132,33.7652,0.0000
C01241=-74.405,-2.621,83.248,178.3277,34.6452,0.0000
C01242=-74.443,0.000,83.276,179.9991,34.6589,0.0000
C01243=-74.405,2.620,83.248,-178.3267,34.6452,0.0000
C01244=-74.307,5.966,83.289,176.7104,33.7645,0.0000
C01245=-75.278,9.949,84.231,165.2926,16.4981,0.0000
C01246=-79.007,11.757,86.605,-178.7272,-0.2829,0.0000
C01247=-85.352,12.799,89.876,-175.7749,-0.7380,0.0000
C01248=-93.717,13.887,93.208,-174.5429,-0.8737,0.0000
C01249=-102.965,15.091,95.718,-173.7590,-0.9993,0.0000
C01250=-111.447,16.532,96.939,-174.1109,-2.0657,0.0000
C01251=-117.648,20.897,97.578,-177.5347,-3.0982,0.0000
C01252=-120.644,27.718,98.094,-179.7087,-1.9012,0.0000
C01253=-119.798,35.596,98.613,179.9644,-0.1215,0.0000
C01254=-117.091,43.748,98.954,179.9948,-0.0139,0.0000
C01255=-113.730,51.862,98.954,179.9938,-0.0135,0.0000
C01256=-109.881,59.540,98.613,179.9393,-0.1111,0.0000
C01257=-104.908,65.708,98.094,178.4495,-1.1387,0.0000
C01258=-97.966,68.413,97.578,176.0690,-0.4486,0.0000
C01259=-90.495,67.115,96.939,174.3778,2.7156,0.0000
C01260=-83.478,62.136,95.718,174.8764,3.7187,0.0000
C01261=-76.088,56.449,93.208,175.5208,3.2492,0.0000
C01262=-69.404,51.303,89.876,176.4895,2.4696,0.0000
C01263=-64.180,47.553,86.605,178.8999,0.7001,0.0000
C01264=-60.264,46.194,84.231,-158.4440,1.3651,0.0000
C01265=-56.761,48.325,83.289,-152.8261,23.3710,0.0000
C01266=-54.465,50.759,83.248,-154.9214,26.9883,0.0000
C01267=-52.639,52.639,83.276,-153.9477,26.0533,0.0000
C01268=-50.759,54.465,83.248,-153.0112,25.0781,0.0000
C01269=-48.325,56.761,83.289,-156.6313,27.1748,0.0000
C01270=-46.194,60.265,84.231,-178.6352,21.5556,0.0000
C01271=-47.553,64.180,86.605,-179.2999,-1.1001,0.0000
C01272=-51.303,69.404,89.876,-177.5304,-3.5105,0.0000
C01273=-56.449,76.088,93.208,-176.7508,-4.4792,0.0000
C01274=-62.136,83.478,95.718,-176.2813,-5.1236,0.0000
C01275=-67.115,90.495,96.939,-177.2844,-5.6222,0.0000
C01276=-68.413,97.966,97.578,179.5514,-3.9310,0.0000
C01277=-65.708,104.908,98.094,178.8613,-1.5505,0.0000
C01278=-59.540,109.881,98.613,179.8889,-0.0607,0.0000
C01279=-51.862,113.730,98.954,179.9865,-0.0062,0.0000
C01280=-43.748,117.091,98.954,179.9861,-0.0052,0.0000
C01281=-35.596,119.798,98.613,179.8785,-0.0356,0.0000
C01282=-27.718,120.644,98.094,178.0988,0.2913,0.0000
C01283=-20.897,117.648,97.578,176.9018,2.4653,0.0000
C01284=-16.532,111.447,96.939,177.9343,5.8891,0.0000
C01285=-15.091,102.965,95.718,179.0007,6.2410,0.0000
C01286=-13.887,93.717,93.208,179.1263,5.4571,0.0000
C01287=-12.799,85.352,89.876,179.2620,4.2251,0.0000
C01288=-11.757,79.007,86.605,179.7171,1.2728,0.0000
C01289=-9.949,75.278,84.231,-163.5019,-14.7074,0.0000
C01290=-5.966,74.307,83.289,-146.2355,-3.2896,0.0000
C01291=-2.620,74.405,83.248,-145.3548,1.6733,0.0000
C01292=0.000,74.443,83.276,-145.3411,-0.0009,0.0000
C01293=0.000,73.205,85.094,-146.1414,-0.0009,0.0000
C01294=2.508,73.170,85.065,-146.1536,-1.5827,0.0000
C01295=5.775,73.084,85.107,-147.0928,3.4640,0.0000
C01296=9.719,74.110,86.081,-164.6300,14.2006,0.0000
C01297=11.485,77.983,88.533,179.6730,-1.5490,0.0000
C01298=12.507,84.540,91.899,179.2973,-4.1637,0.0000
C01299=13.596,93.149,95.314,179.1887,-5.2120,0.0000
C01300=14.803,102.622,97.872,179.0896,-5.8667,0.0000
C01301=16.233,111.284,99.113,178.1114,-5.5113,0.0000
C01302=20.622,117.615,99.760,177.1245,-2.3209,0.0000
C01303=27.505,120.682,100.284,178.2326,-0.2776,0.0000
C01304=35.464,119.842,100.809,179.8870,0.0331,0.0000
C01305=43.704,117.108,101.154,179.9871,0.0048,0.0000
C01306=51.905,113.711,101.154,179.9875,0.0057,0.0000
C01307=59.664,109.818,100.809,179.8967,0.0565,0.0000
C01308=65.886,104.784,100.284,178.9463,1.4461,0.0000
C01309=68.584,97.748,99.760,179.6070,3.6720,0.0000
C01310=67.211,90.168,99.113,-177.4285,5.2304,0.0000
C01311=62.097,83.032,97.872,-176.4853,4.7955,0.0000
C01312=56.252,75.480,95.314,-176.8812,4.2615,0.0000
C01313=50.935,68.623,91.899,-177.5490,3.4422,0.0000
C01314=47.021,63.263,88.533,-179.1357,1.3266,0.0000
C01315=45.531,59.276,86.081,-179.1156,-20.4708,0.0000
C01316=47.594,55.761,85.107,-157.4728,-26.5823,0.0000
C01317=49.966,53.512,85.065,-153.7229,-24.4493,0.0000
C01318=51.764,51.764,85.094,-154.6191,-25.3798,0.0000
C01319=53.512,49.966,85.065,-155.5512,-26.2777,0.0000
C01320=55.762,47.594,85.108,-153.4168,-22.5249,0.0000
C01321=59.276,45.531,86.082,-159.5296,-0.8841,0.0000
C01322=63.263,47.021,88.533,178.6734,-0.8643,0.0000
C01323=68.623,50.935,91.899,176.5578,-2.4510,0.0000
C01324=75.480,56.252,95.314,175.7385,-3.1188,0.0000
C01325=83.032,62.097,97.872,175.2045,-3.5147,0.0000
C01326=90.168,67.211,99.113,174.7696,-2.5715,0.0000
C01327=97.748,68.584,99.760,176.3280,0.3930,0.0000
C01328=104.784,65.886,100.284,178.5539,1.0537,0.0000
C01329=109.818,59.664,100.809,179.9435,0.1033,0.0000
C01330=113.711,51.905,101.154,179.9943,0.0125,0.0000
C01331=117.108,43.704,101.154,179.9952,0.0129,0.0000
C01332=119.842,35.464,100.809,179.9669,0.1130,0.0000
C01333=120.682,27.505,100.284,-179.7224,1.7674,0.0000
C01334=117.615,20.622,99.760,-177.6791,2.8755,0.0000
C01335=111.284,16.233,99.113,-174.4887,1.8886,0.0000
C01336=102.622,14.803,97.872,-174.1333,0.9104,0.0000
C01337=93.149,13.596,95.314,-174.7880,0.8113,0.0000
C01338=84.540,12.507,91.899,-175.8363,0.7027,0.0000
C01339=77.983,11.485,88.533,-178.4510,0.3270,0.0000
C01340=74.110,9.719,86.081,165.7994,-15.3700,0.0000
C01341=73.084,5.775,85.107,176.5360,-32.9072,0.0000
C01342=73.170,2.508,85.065,-178.4173,-33.8464,0.0000
C01343=73.205,0.000,85.094,-179.9991,-33.8586,0.0000
C01344=73.170,-2.507,85.065,178.4163,-33.8464,0.0000
C01345=73.084,-5.775,85.108,-176.5333,-32.9064,0.0000
C01346=74.110,-9.719,86.082,-165.7995,-15.3694,0.0000
C01347=77.983,-11.485,88.533,178.4510,0.3270,0.0000
C01348=84.540,-12.507,91.899,175.8363,0.7027,0.0000
C01349=93.149,-13.596,95.314,174.7880,0.8113,0.0000
C01350=102.622,-14.803,97.872,174.1333,0.9104,0.0000
C01351=111.284,-16.233,99.113,174.4887,1.8886,0.0000
C01352=117.615,-20.622,99.760,177.6791,2.8755,0.0000
C01353=120.682,-27.505,100.284,179.7224,1.7674,0.0000
C01354=119.842,-35.464,100.809,-179.9669,0.1130,0.0000
C01355=117.108,-43.704,101.154,-179.9952,0.0129,0.0000
C01356=113.711,-51.905,101.154,-179.9943,0.0125,0.0000
C01357=109.818,-59.664,100.809,-179.9435,0.1033,0.0000
C01358=104.784,-65.886,100.284,-178.5539,1.0537,0.0000
C01359=97.748,-68.584,99.760,-176.3280,0.3930,0.0000
C01360=90.168,-67.211,99.113,-174.7696,-2.5715,0.0000
C01361=83.032,-62.097,97.872,-175.2045,-3.5147,0.0000
C01362=75.480,-56.252,95.314,-175.7385,-3.1188,0.0000
C01363=68.623,-50.935,91.899,-176.5578,-2.4510,0.0000
C01364=63.263,-47.021,88.533,-178.6734,-0.8643,0.0000
C01365=59.276,-45.531,86.081,159.5292,-0.8844,0.0000
C01366=55.761,-47.594,85.107,153.4177,-22.5272,0.0000
C01367=53.512,-49.966,85.065,155.5507,-26.2771,0.0000
C01368=51.764,-51.764,85.094,154.6202,-25.3809,0.0000
C01369=49.966,-53.512,85.065,153.7223,-24.4488,0.0000
C01370=47.594,-55.762,85.108,157.4751,-26.5832,0.0000
C01371=45.531,-59.276,86.082,179.1159,-20.4704,0.0000
C01372=47.021,-63.263,88.533,179.1357,1.3266,0.0000
C01373=50.935,-68.623,91.899,177.5490,3.4422,0.0000
C01374=56.252,-75.480,95.314,176.8812,4.2615,0.0000
C01375=62.097,-83.032,97.872,176.4853,4.7955,0.0000
C01376=67.211,-90.168,99.113,177.4285,5.2304,0.0000
C01377=68.584,-97.748,99.760,-179.6070,3.6720,0.0000
C01378=65.886,-104.784,100.284,-178.9463,1.4461,0.0000
C01379=59.664,-109.818,100.809,-179.8967,0.0565,0.0000
C01380=51.905,-113.711,101.154,-179.9875,0.0057,0.0000
C01381=43.704,-117.108,101.154,-179.9871,0.0048,0.0000
C01382=35.464,-119.842,100.809,-179.8870,0.0331,0.0000
C01383=27.505,-120.682,100.284,-178.2326,-0.2776,0.0000
C01384=20.622,-117.615,99.760,-177.1245,-2.3209,0.0000
C01385=16.233,-111.284,99.113,-178.1114,-5.5113,0.0000
C01386=14.803,-102.622,97.872,-179.0896,-5.8667,0.0000
C01387=13.596,-93.149,95.314,-179.1887,-5.2120,0.0000
C01388=12.507,-84.540,91.899,-179.2973,-4.1637,0.0000
C01389=11.485,-77.983,88.533,-179.6730,-1.5490,0.0000
C01390=9.719,-74.110,86.081,164.6300,14.2006,0.0000
C01391=5.775,-73.084,85.107,147.0928,3.4640,0.0000
C01392=2.508,-73.170,85.065,146.1536,-1.5827,0.0000
C01393=0.000,-73.205,85.094,146.1414,-0.0009,0.0000
C01394=0.000,-73.205,85.094,146.1414,-0.0009,0.0000
C01395=-2.507,-73.170,85.065,146.1536,1.5837,0.0000
C01396=-5.775,-73.084,85.108,147.0936,-3.4667,0.0000
C01397=-9.719,-74.110,86.082,164.6306,-14.2005,0.0000
C01398=-11.485,-77.983,88.533,-179.6730,1.5490,0.0000
C01399=-12.507,-84.540,91.899,-179.2973,4.1637,0.0000
C01400=-13.596,-93.149,95.314,-179.1887,5.2120,0.0000
C01401=-14.803,-102.622,97.872,-179.0896,5.8667,0.0000
C01402=-16.233,-111.284,99.113,-178.1114,5.5113,0.0000
C01403=-20.622,-117.615,99.760,-177.1245,2.3209,0.0000
C01404=-27.505,-120.682,100.284,-178.2326,0.2776,0.0000
C01405=-35.464,-119.842,100.809,-179.8870,-0.0331,0.0000
C01406=-43.704,-117.108,101.154,-179.9871,-0.0048,0.0000
C01407=-51.905,-113.711,101.154,-179.9875,-0.0057,0.0000
C01408=-59.664,-109.818,100.809,-179.8967,-0.0565,0.0000
C01409=-65.886,-104.784,100.284,-178.9463,-1.4461,0.0000
C01410=-68.584,-97.748,99.760,-179.6070,-3.6720,0.0000
C01411=-67.211,-90.168,99.113,177.4285,-5.2304,0.0000
C01412=-62.097,-83.032,97.872,176.4853,-4.7955,0.0000
C01413=-56.252,-75.480,95.314,176.8812,-4.2615,0.0000
C01414=-50.935,-68.623,91.899,177.5490,-3.4422,0.0000
C01415=-47.021,-63.263,88.533,179.1357,-1.3266,0.0000
C01416=-45.531,-59.276,86.081,179.1156,20.4708,0.0000
C01417=-47.594,-55.761,85.107,157.4728,26.5823,0.0000
C01418=-49.966,-53.512,85.065,153.7229,24.4493,0.0000
C01419=-51.764,-51.764,85.094,154.6191,25.3798,0.0000
C01420=-53.512,-49.966,85.065,155.5512,26.2777,0.0000
C01421=-55.762,-47.594,85.108,153.4168,22.5249,0.0000
C01422=-59.276,-45.531,86.082,159.5296,0.8841,0.0000
C01423=-63.263,-47.021,88.533,-178.6734,0.8643,0.0000
C01424=-68.623,-50.935,91.899,-176.5578,2.4510,0.0000
C01425=-75.480,-56.252,95.314,-175.7385,3.1188,0.0000
C01426=-83.032,-62.097,97.872,-175.2045,3.5147,0.0000
C01427=-90.168,-67.211,99.113,-174.7696,2.5715,0.0000
C01428=-97.748,-68.584,99.760,-176.3280,-0.3930,0.0000
C01429=-104.784,-65.886,100.284,-178.5539,-1.0537,0.0000
C01430=-109.818,-59.664,100.809,-179.9435,-0.1033,0.0000
C01431=-113.711,-51.905,101.154,-179.9943,-0.0125,0.0000
C01432=-117.108,-43.704,101.154,-179.9952,-0.0129,0.0000
C01433=-119.842,-35.464,100.809,-179.9669,-0.1130,0.0000
C01434=-120.682,-27.505,100.284,179.7224,-1.7674,0.0000
C01435=-117.615,-20.622,99.760,177.6791,-2.8755,0.0000
C01436=-111.284,-16.233,99.113,174.4887,-1.8886,0.0000
C01437=-102.622,-14.803,97.872,174.1333,-0.9104,0.0000
C01438=-93.149,-13.596,95.314,174.7880,-0.8113,0.0000
C01439=-84.540,-12.507,91.899,175.8363,-0.7027,0.0000
C01440=-77.983,-11.485,88.533,178.4510,-0.3270,0.0000
C01441=-74.110,-9.719,86.081,-165.7994,15.3700,0.0000
C01442=-73.084,-5.775,85.107,-176.5360,32.9072,0.0000
C01443=-73.170,-2.508,85.065,178.4173,33.8464,0.0000
C01444=-73.205,0.000,85.094,179.9991,33.8586,0.0000
C01445=-73.170,2.507,85.065,-178.4163,33.8464,0.0000
C01446=-73.084,5.775,85.108,176.5333,32.9064,0.0000
C01447=-74.110,9.719,86.082,165.7995,15.3694,0.0000
C01448=-77.983,11.485,88.533,-178.4510,-0.3270,0.0000
C01449=-84.540,12.507,91.899,-175.8363,-0.7027,0.0000
C01450=-93.149,13.596,95.314,-174.7880,-0.8113,0.0000
C01451=-102.622,14.803,97.872,-174.1333,-0.9104,0.0000
C01452=-111.284,16.233,99.113,-174.4887,-1.8886,0.0000
C01453=-117.615,20.622,99.760,-177.6791,-2.8755,0.0000
C01454=-120.682,27.505,100.284,-179.7224,-1.7674,0.0000
C01455=-119.842,35.464,100.809,179.9669,-0.1130,0.0000
C01456=-117.108,43.704,101.154,179.9952,-0.0129,0.0000
C01457=-113.711,51.905,101.154,179.9943,-0.0125,0.0000
C01458=-109.818,59.664,100.809,179.9435,-0.1033,0.0000
C01459=-104.784,65.886,100.284,178.5539,-1.0537,0.0000
C01460=-97.748,68.584,99.760,176.3280,-0.3930,0.0000
C01461=-90.168,67.211,99.113,174.7696,2.5715,0.0000
C01462=-83.032,62.097,97.872,175.2045,3.5147,0.0000
C01463=-75.480,56.252,95.314,175.7385,3.1188,0.0000
C01464=-68.623,50.935,91.899,176.5578,2.4510,0.0000
C01465=-63.263,47.021,88.533,178.6734,0.8643,0.0000
C01466=-59.276,45.531,86.081,-159.5292,0.8844,0.0000
C01467=-55.761,47.594,85.107,-153.4177,22.5272,0.0000
C01468=-53.512,49.966,85.065,-155.5507,26.2771,0.0000
C01469=-51.764,51.764,85.094,-154.6202,25.3809,0.0000
C01470=-49.966,53.512,85.065,-153.7223,24.4488,0.0000
C01471=-47.594,55.762,85.108,-157.4751,26.5832,0.0000
C01472=-45.531,59.276,86.082,-179.1159,20.4704,0.0000
C01473=-47.021,63.263,88.533,-179.1357,-1.3266,0.0000
C01474=-50.935,68.623,91.899,-177.5490,-3.4422,0.0000
C01475=-56.252,75.480,95.314,-176.8812,-4.2615,0.0000
C01476=-62.097,83.032,97.872,-176.4853,-4.7955,0.0000
C01477=-67.211,90.168,99.113,-177.4285,-5.2304,0.0000
C01478=-68.584,97.748,99.760,179.6070,-3.6720,0.0000
C01479=-65.886,104.784,100.284,178.9463,-1.4461,0.0000
C01480=-59.664,109.818,100.809,179.8967,-0.0565,0.0000
C01481=-51.905,113.711,101.154,179.9875,-0.0057,0.0000
C01482=-43.704,117.108,101.154,179.9871,-0.0048,0.0000
C01483=-35.464,119.842,100.809,179.8870,-0.0331,0.0000
C01484=-27.505,120.682,100.284,178.2326,0.2776,0.0000
C01485=-20.622,117.615,99.760,177.1245,2.3209,0.0000
C01486=-16.233,111.284,99.113,178.1114,5.5113,0.0000
C01487=-14.803,102.622,97.872,179.0896,5.8667,0.0000
C01488=-13.596,93.149,95.314,179.1887,5.2120,0.0000
C01489=-12.507,84.540,91.899,179.2973,4.1637,0.0000
C01490=-11.485,77.983,88.533,179.6730,1.5490,0.0000
C01491=-9.719,74.110,86.082,-164.6306,-14.2005,0.0000
C01492=-5.775,73.084,85.108,-147.0936,-3.4667,0.0000
C01493=-2.507,73.170,85.065,-146.1536,1.5837,0.0000
C01494=0.000,73.205,85.094,-146.1414,-0.0009,0.0000
C01495=0.000,71.993,86.930,-147.0265,-0.0009,0.0000
C01496=2.397,71.962,86.901,-147.0370,-1.4892,0.0000
C01497=5.589,71.887,86.944,-148.0352,3.6143,0.0000
C01498=9.494,72.971,87.950,-165.7390,13.6389,0.0000
C01499=11.222,76.989,90.478,179.6440,-1.7725,0.0000
C01500=12.227,83.762,93.938,179.3362,-4.0634,0.0000
C01501=13.321,92.612,97.429,179.2524,-4.9303,0.0000
C01502=14.535,102.303,100.032,179.1779,-5.4532,0.0000
C01503=15.957,111.134,101.290,178.2918,-5.0922,0.0000
C01504=20.370,117.584,101.945,177.3660,-2.1532,0.0000
C01505=27.310,120.718,102.475,178.3801,-0.2600,0.0000
C01506=35.344,119.882,103.005,179.8965,0.0302,0.0000
C01507=43.664,117.124,103.353,179.9882,0.0044,0.0000
C01508=51.944,113.694,103.353,179.9886,0.0052,0.0000
C01509=59.777,109.761,103.005,179.9054,0.0518,0.0000
C01510=66.049,104.671,102.475,179.0382,1.3294,0.0000
C01511=68.741,97.548,101.945,179.6595,3.3832,0.0000
C01512=67.300,89.867,101.290,-177.5994,4.8072,0.0000
C01513=62.061,82.617,100.032,-176.7173,4.4401,0.0000
C01514=56.067,74.906,97.429,-177.0365,4.0169,0.0000
C01515=50.583,67.875,93.938,-177.5927,3.3436,0.0000
C01516=46.505,62.375,90.478,-178.9981,1.5052,0.0000
C01517=44.885,58.312,87.950,-179.5330,-19.3565,0.0000
C01518=46.880,54.783,86.944,-158.3677,-25.9156,0.0000
C01519=49.190,52.579,86.901,-154.5019,-23.7576,0.0000
C01520=50.907,50.907,86.930,-155.3568,-24.6421,0.0000
C01521=52.579,49.190,86.901,-156.2430,-25.4987,0.0000
C01522=54.784,46.880,86.944,-154.0835,-21.6299,0.0000
C01523=58.312,44.885,87.950,-160.6440,-0.4666,0.0000
C01524=62.375,46.505,90.478,178.4948,-1.0019,0.0000
C01525=67.875,50.583,93.938,176.6564,-2.4073,0.0000
C01526=74.906,56.067,97.429,175.9831,-2.9635,0.0000
C01527=82.617,62.061,100.032,175.5599,-3.2827,0.0000
C01528=89.867,67.300,101.290,175.1928,-2.4006,0.0000
C01529=97.548,68.741,101.945,176.6168,0.3405,0.0000
C01530=104.671,66.049,102.475,178.6706,0.9618,0.0000
C01531=109.761,59.777,103.005,179.9482,0.0946,0.0000
C01532=113.694,51.944,103.353,179.9948,0.0114,0.0000
C01533=117.124,43.664,103.353,179.9956,0.0118,0.0000
C01534=119.882,35.344,103.005,179.9698,0.1035,0.0000
C01535=120.718,27.310,102.475,-179.7400,1.6199,0.0000
C01536=117.584,20.370,101.945,-177.8468,2.6340,0.0000
C01537=111.134,15.957,101.290,-174.9078,1.7082,0.0000
C01538=102.303,14.535,100.032,-174.5468,0.8221,0.0000
C01539=92.612,13.321,97.429,-175.0697,0.7476,0.0000
C01540=83.762,12.227,93.938,-175.9366,0.6638,0.0000
C01541=76.989,11.222,90.478,-178.2275,0.3560,0.0000
C01542=72.971,9.494,87.950,166.3611,-14.2610,0.0000
C01543=71.887,5.589,86.944,176.3857,-31.9648,0.0000
C01544=71.962,2.397,86.901,-178.5108,-32.9630,0.0000
C01545=71.993,0.000,86.930,-179.9991,-32.9735,0.0000
C01546=71.962,-2.396,86.901,178.5098,-32.9630,0.0000
C01547=71.887,-5.589,86.944,-176.3830,-31.9640,0.0000
C01548=72.971,-9.494,87.950,-166.3612,-14.2604,0.0000
C01549=76.989,-11.222,90.478,178.2275,0.3560,0.0000
C01550=83.762,-12.227,93.938,175.9366,0.6638,0.0000
C01551=92.612,-13.321,97.429,175.0697,0.7476,0.0000
C01552=102.303,-14.535,100.032,174.5468,0.8221,0.0000
C01553=111.134,-15.957,101.290,174.9078,1.7082,0.0000
C01554=117.584,-20.370,101.945,177.8468,2.6340,0.0000
C01555=120.718,-27.310,102.475,179.7400,1.6199,0.0000
C01556=119.882,-35.344,103.005,-179.9698,0.1035,0.0000
C01557=117.124,-43.664,103.353,-179.9956,0.0118,0.0000
C01558=113.694,-51.944,103.353,-179.9948,0.0114,0.0000
C01559=109.761,-59.777,103.005,-179.9482,0.0946,0.0000
C01560=104.671,-66.049,102.475,-178.6706,0.9618,0.0000
C01561=97.548,-68.741,101.945,-176.6168,0.3405,0.0000
C01562=89.867,-67.300,101.290,-175.1928,-2.4006,0.0000
C01563=82.617,-62.061,100.032,-175.5599,-3.2827,0.0000
C01564=74.906,-56.067,97.429,-175.9831,-2.9635,0.0000
C01565=67.875,-50.583,93.938,-176.6564,-2.4073,0.0000
C01566=62.375,-46.505,90.478,-178.4948,-1.0019,0.0000
C01567=58.312,-44.885,87.950,160.6435,-0.4670,0.0000
C01568=54.783,-46.880,86.944,154.0844,-21.6323,0.0000
C01569=52.579,-49.190,86.901,156.2424,-25.4981,0.0000
C01570=50.907,-50.907,86.930,155.3579,-24.6432,0.0000
C01571=49.190,-52.579,86.901,154.5013,-23.7570,0.0000
C01572=46.880,-54.784,86.944,158.3701,-25.9165,0.0000
C01573=44.885,-58.312,87.950,179.5334,-19.3560,0.0000
C01574=46.505,-62.375,90.478,178.9981,1.5052,0.0000
C01575=50.583,-67.875,93.938,177.5927,3.3436,0.0000
C01576=56.067,-74.906,97.429,177.0365,4.0169,0.0000
C01577=62.061,-82.617,100.032,176.7173,4.4401,0.0000
C01578=67.300,-89.867,101.290,177.5994,4.8072,0.0000
C01579=68.741,-97.548,101.945,-179.6595,3.3832,0.0000
C01580=66.049,-104.671,102.475,-179.0382,1.3294,0.0000
C01581=59.777,-109.761,103.005,-179.9054,0.0518,0.0000
C01582=51.944,-113.694,103.353,-179.9886,0.0052,0.0000
C01583=43.664,-117.124,103.353,-179.9882,0.0044,0.0000
C01584=35.344,-119.882,103.005,-179.8965,0.0302,0.0000
C01585=27.310,-120.718,102.475,-178.3801,-0.2600,0.0000
C01586=20.370,-117.584,101.945,-177.3660,-2.1532,0.0000
C01587=15.957,-111.134,101.290,-178.2918,-5.0922,0.0000
C01588=14.535,-102.303,100.032,-179.1779,-5.4532,0.0000
C01589=13.321,-92.612,97.429,-179.2524,-4.9303,0.0000
C01590=12.227,-83.762,93.938,-179.3362,-4.0634,0.0000
C01591=11.222,-76.989,90.478,-179.6440,-1.7725,0.0000
C01592=9.494,-72.971,87.950,165.7390,13.6389,0.0000
C01593=5.589,-71.887,86.944,148.0352,3.6143,0.0000
C01594=2.397,-71.962,86.901,147.0370,-1.4892,0.0000
C01595=0.000,-71.993,86.930,147.0265,-0.0009,0.0000
C01596=0.000,-71.993,86.930,147.0265,-0.0009,0.0000
C01597=-2.396,-71.962,86.901,147.0370,1.4902,0.0000
C01598=-5.589,-71.887,86.944,148.0360,-3.6170,0.0000
C01599=-9.494,-72.971,87.950,165.7396,-13.6388,0.0000
C01600=-11.222,-76.989,90.478,-179.6440,1.7725,0.0000
C01601=-12.227,-83.762,93.938,-179.3362,4.0634,0.0000
C01602=-13.321,-92.612,97.429,-179.2524,4.9303,0.0000
C01603=-14.535,-102.303,100.032,-179.1779,5.4532,0.0000
C01604=-15.957,-111.134,101.290,-178.2918,5.0922,0.0000
C01605=-20.370,-117.584,101.945,-177.3660,2.1532,0.0000
C01606=-27.310,-120.718,102.475,-178.3801,0.2600,0.0000
C01607=-35.344,-119.882,103.005,-179.8965,-0.0302,0.0000
C01608=-43.664,-117.124,103.353,-179.9882,-0.0044,0.0000
C01609=-51.944,-113.694,103.353,-179.9886,-0.0052,0.0000
C01610=-59.777,-109.761,103.005,-179.9054,-0.0518,0.0000
C01611=-66.049,-104.671,102.475,-179.0382,-1.3294,0.0000
C01612=-68.741,-97.548,101.945,-179.6595,-3.3832,0.0000
C01613=-67.300,-89.867,101.290,177.5994,-4.8072,0.0000
C01614=-62.061,-82.617,100.032,176.7173,-4.4401,0.0000
C01615=-56.067,-74.906,97.429,177.0365,-4.0169,0.0000
C01616=-50.583,-67.875,93.938,177.5927,-3.3436,0.0000
C01617=-46.505,-62.375,90.478,178.9981,-1.5052,0.0000
C01618=-44.885,-58.312,87.950,179.5330,19.3565,0.0000
C01619=-46.880,-54.783,86.944,158.3677,25.9156,0.0000
C01620=-49.190,-52.579,86.901,154.5019,23.7576,0.0000
C01621=-50.907,-50.907,86.930,155.3568,24.6421,0.0000
C01622=-52.579,-49.190,86.901,156.2430,25.4987,0.0000
C01623=-54.784,-46.880,86.944,154.0835,21.6299,0.0000
C01624=-58.312,-44.885,87.950,160.6440,0.4666,0.0000
C01625=-62.375,-46.505,90.478,-178.4948,1.0019,0.0000
C01626=-67.875,-50.583,93.938,-176.6564,2.4073,0.0000
C01627=-74.906,-56.067,97.429,-175.9831,2.9635,0.0000
C01628=-82.617,-62.061,100.032,-175.5599,3.2827,0.0000
C01629=-89.867,-67.300,101.290,-175.1928,2.4006,0.0000
C01630=-97.548,-68.741,101.945,-176.6168,-0.3405,0.0000
C01631=-104.671,-66.049,102.475,-178.6706,-0.9618,0.0000
C01632=-109.761,-59.777,103.005,-179.9482,-0.0946,0.0000
C01633=-113.694,-51.944,103.353,-179.9948,-0.0114,0.0000
C01634=-117.124,-43.664,103.353,-179.9956,-0.0118,0.0000
C01635=-119.882,-35.344,103.005,-179.9698,-0.1035,0.0000
C01636=-120.718,-27.310,102.475,179.7400,-1.6199,0.0000
C01637=-117.584,-20.370,101.945,177.8468,-2.6340,0.0000
C01638=-111.134,-15.957,101.290,174.9078,-1.7082,0.0000
C01639=-102.303,-14.535,100.032,174.5468,-0.8221,0.0000
C01640=-92.612,-13.321,97.429,175.0697,-0.7476,0.0000
C01641=-83.762,-12.227,93.938,175.9366,-0.6638,0.0000
C01642=-76.989,-11.222,90.478,178.2275,-0.3560,0.0000
C01643=-72.971,-9.494,87.950,-166.3611,14.2610,0.0000
C01644=-71.887,-5.589,86.944,-176.3857,31.9648,0.0000
C01645=-71.962,-2.397,86.901,178.5108,32.9630,0.0000
C01646=-71.993,0.000,86.930,179.9991,32.9735,0.0000
C01647=-71.962,2.396,86.901,-178.5098,32.9630,0.0000
C01648=-71.887,5.589,86.944,176.3830,31.9640,0.0000
C01649=-72.971,9.494,87.950,166.3612,14.2604,0.0000
C01650=-76.989,11.222,90.478,-178.2275,-0.3560,0.0000
C01651=-83.762,12.227,93.938,-175.9366,-0.6638,0.0000
C01652=-92.612,13.321,97.429,-175.0697,-0.7476,0.0000
C01653=-102.303,14.535,100.032,-174.5468,-0.8221,0.0000
C01654=-111.134,15.957,101.290,-174.9078,-1.7082,0.0000
C01655=-117.584,20.370,101.945,-177.8468,-2.6340,0.0000
C01656=-120.718,27.310,102.475,-179.7400,-1.6199,0.0000
C01657=-119.882,35.344,103.005,179.9698,-0.1035,0.0000
C01658=-117.124,43.664,103.353,179.9956,-0.0118,0.0000
C01659=-113.694,51.944,103.353,179.9948,-0.0114,0.0000
C01660=-109.761,59.777,103.005,179.9482,-0.0946,0.0000
C01661=-104.671,66.049,102.475,178.6706,-0.9618,0.0000
C01662=-97.548,68.741,101.945,176.6168,-0.3405,0.0000
C01663=-89.867,67.300,101.290,175.1928,2.4006,0.0000
C01664=-82.617,62.061,100.032,175.5599,3.2827,0.0000
C01665=-74.906,56.067,97.429,175.9831,2.9635,0.0000
C01666=-67.875,50.583,93.938,176.6564,2.4073,0.0000
C01667=-62.375,46.505,90.478,178.4948,1.0019,0.0000
C01668=-58.312,44.885,87.950,-160.6435,0.4670,0.0000
C01669=-54.783,46.880,86.944,-154.0844,21.6323,0.0000
C01670=-52.579,49.190,86.901,-156.2424,25.4981,0.0000
C01671=-50.907,50.907,86.930,-155.3579,24.6432,0.0000
C01672=-49.190,52.579,86.901,-154.5013,23.7570,0.0000
C01673=-46.880,54.784,86.944,-158.3701,25.9165,0.0000
C01674=-44.885,58.312,87.950,-179.5334,19.3560,0.0000
C01675=-46.505,62.375,90.478,-178.9981,-1.5052,0.0000
C01676=-50.583,67.875,93.938,-177.5927,-3.3436,0.0000
C01677=-56.067,74.906,97.429,-177.0365,-4.0169,0.0000
C01678=-62.061,82.617,100.032,-176.7173,-4.4401,0.0000
C01679=-67.300,89.867,101.290,-177.5994,-4.8072,0.0000
C01680=-68.741,97.548,101.945,179.6595,-3.3832,0.0000
C01681=-66.049,104.671,102.475,179.0382,-1.3294,0.0000
C01682=-59.777,109.761,103.005,179.9054,-0.0518,0.0000
C01683=-51.944,113.694,103.353,179.9886,-0.0052,0.0000
C01684=-43.664,117.124,103.353,179.9882,-0.0044,0.0000
C01685=-35.344,119.882,103.005,179.8965,-0.0302,0.0000
C01686=-27.310,120.718,102.475,178.3801,0.2600,0.0000
C01687=-20.370,117.584,101.945,177.3660,2.1532,0.0000
C01688=-15.957,111.134,101.290,178.2918,5.0922,0.0000
C01689=-14.535,102.303,100.032,179.1779,5.4532,0.0000
C01690=-13.321,92.612,97.429,179.2524,4.9303,0.0000
C01691=-12.227,83.762,93.938,179.3362,4.0634,0.0000
C01692=-11.222,76.989,90.478,179.6440,1.7725,0.0000
C01693=-9.494,72.971,87.950,-165.7396,-13.6388,0.0000
C01694=-5.589,71.887,86.944,-148.0360,-3.6170,0.0000
C01695=-2.396,71.962,86.901,-147.0370,1.4902,0.0000
C01696=0.000,71.993,86.930,-147.0265,-0.0009,0.0000
C01697=0.000,70.811,88.785,-148.0029,-0.0009,0.0000
C01698=2.289,70.783,88.755,-148.0116,-1.3922,0.0000
C01699=5.407,70.720,88.800,-149.0673,3.7344,0.0000
C01700=9.276,71.863,89.838,-166.8248,13.0264,0.0000
C01701=10.968,76.031,92.442,179.6279,-1.9440,0.0000
C01702=11.961,83.022,95.993,179.3784,-3.9245,0.0000
C01703=13.065,92.111,99.556,179.3173,-4.6124,0.0000
C01704=14.289,102.010,102.199,179.2658,-5.0011,0.0000
C01705=15.705,110.997,103.471,178.4754,-4.6328,0.0000
C01706=20.141,117.557,104.133,177.6257,-1.9629,0.0000
C01707=27.134,120.750,104.667,178.5409,-0.2387,0.0000
C01708=35.236,119.917,105.202,179.9070,0.0271,0.0000
C01709=43.628,117.138,105.553,179.9895,0.0039,0.0000
C01710=51.979,113.678,105.553,179.9898,0.0047,0.0000
C01711=59.878,109.710,105.202,179.9151,0.0466,0.0000
C01712=66.196,104.570,104.667,179.1369,1.2005,0.0000
C01713=68.883,97.367,104.133,179.7087,3.0654,0.0000
C01714=67.381,89.592,103.471,-177.7964,4.3530,0.0000
C01715=62.028,82.235,102.199,-176.9767,4.0577,0.0000
C01716=55.894,74.370,99.556,-177.2164,3.7459,0.0000
C01717=50.248,67.163,95.993,-177.6615,3.2156,0.0000
C01718=46.007,61.518,92.442,-178.8881,1.6378,0.0000
C01719=44.256,57.374,89.838,-179.8891,-18.2174,0.0000
C01720=46.183,53.830,88.800,-159.3140,-25.1687,0.0000
C01721=48.433,51.670,88.755,-155.3527,-22.9995,0.0000
C01722=50.071,50.071,88.785,-156.1636,-23.8353,0.0000
C01723=51.669,48.433,88.755,-157.0010,-24.6479,0.0000
C01724=53.830,46.183,88.800,-154.8304,-20.6837,0.0000
C01725=57.374,44.256,89.838,-161.7832,-0.1105,0.0000
C01726=61.518,46.007,92.442,178.3622,-1.1119,0.0000
C01727=67.163,50.248,95.993,176.7844,-2.3385,0.0000
C01728=74.370,55.894,99.556,176.2541,-2.7836,0.0000
C01729=82.235,62.028,102.199,175.9423,-3.0233,0.0000
C01730=89.592,67.381,103.471,175.6470,-2.2036,0.0000
C01731=97.367,68.883,104.133,176.9346,0.2913,0.0000
C01732=104.570,66.196,104.667,178.7995,0.8631,0.0000
C01733=109.710,59.878,105.202,179.9534,0.0849,0.0000
C01734=113.678,51.979,105.553,179.9953,0.0102,0.0000
C01735=117.138,43.628,105.553,179.9961,0.0105,0.0000
C01736=119.917,35.236,105.202,179.9729,0.0930,0.0000
C01737=120.750,27.134,104.667,-179.7613,1.4591,0.0000
C01738=117.557,20.141,104.133,-178.0371,2.3743,0.0000
C01739=110.997,15.705,103.471,-175.3672,1.5246,0.0000
C01740=102.010,14.289,102.199,-174.9989,0.7342,0.0000
C01741=92.111,13.065,99.556,-175.3876,0.6827,0.0000
C01742=83.022,11.961,95.993,-176.0755,0.6216,0.0000
C01743=76.031,10.968,92.442,-178.0560,0.3721,0.0000
C01744=71.863,9.276,89.838,166.9736,-13.1752,0.0000
C01745=70.720,5.407,88.800,176.2656,-30.9327,0.0000
C01746=70.783,2.289,88.755,-178.6078,-31.9884,0.0000
C01747=70.811,0.000,88.785,-179.9991,-31.9971,0.0000
C01748=70.783,-2.288,88.755,178.6068,-31.9884,0.0000
C01749=70.720,-5.408,88.800,-176.2629,-30.9319,0.0000
C01750=71.863,-9.276,89.838,-166.9737,-13.1745,0.0000
C01751=76.031,-10.968,92.442,178.0560,0.3721,0.0000
C01752=83.022,-11.961,95.993,176.0755,0.6216,0.0000
C01753=92.111,-13.065,99.556,175.3876,0.6827,0.0000
C01754=102.010,-14.289,102.199,174.9989,0.7342,0.0000
C01755=110.997,-15.705,103.471,175.3672,1.5246,0.0000
C01756=117.557,-20.141,104.133,178.0371,2.3743,0.0000
C01757=120.750,-27.134,104.667,179.7613,1.4591,0.0000
C01758=119.917,-35.236,105.202,-179.9729,0.0930,0.0000
C01759=117.138,-43.628,105.553,-179.9961,0.0105,0.0000
C01760=113.678,-51.979,105.553,-179.9953,0.0102,0.0000
C01761=109.710,-59.878,105.202,-179.9534,0.0849,0.0000
C01762=104.570,-66.196,104.667,-178.7995,0.8631,0.0000
C01763=97.367,-68.883,104.133,-176.9346,0.2913,0.0000
C01764=89.592,-67.381,103.471,-175.6470,-2.2036,0.0000
C01765=82.235,-62.028,102.199,-175.9423,-3.0233,0.0000
C01766=74.370,-55.894,99.556,-176.2541,-2.7836,0.0000
C01767=67.163,-50.248,95.993,-176.7844,-2.3385,0.0000
C01768=61.518,-46.007,92.442,-178.3622,-1.1119,0.0000
C01769=57.374,-44.256,89.838,161.7826,-0.1109,0.0000
C01770=53.830,-46.183,88.800,154.8313,-20.6860,0.0000
C01771=51.670,-48.433,88.755,157.0005,-24.6473,0.0000
C01772=50.071,-50.071,88.785,156.1647,-23.8364,0.0000
C01773=48.433,-51.669,88.755,155.3521,-22.9990,0.0000
C01774=46.183,-53.830,88.800,159.3163,-25.1696,0.0000
C01775=44.256,-57.374,89.838,179.8895,-18.2168,0.0000
C01776=46.007,-61.518,92.442,178.8881,1.6378,0.0000
C01777=50.248,-67.163,95.993,177.6615,3.2156,0.0000
C01778=55.894,-74.370,99.556,177.2164,3.7459,0.0000
C01779=62.028,-82.235,102.199,176.9767,4.0577,0.0000
C01780=67.381,-89.592,103.471,177.7964,4.3530,0.0000
C01781=68.883,-97.367,104.133,-179.7087,3.0654,0.0000
C01782=66.196,-104.570,104.667,-179.1369,1.2005,0.0000
C01783=59.878,-109.710,105.202,-179.9151,0.0466,0.0000
C01784=51.979,-113.678,105.553,-179.9898,0.0047,0.0000
C01785=43.628,-117.138,105.553,-179.9895,0.0039,0.0000
C01786=35.236,-119.917,105.202,-179.9070,0.0271,0.0000
C01787=27.134,-120.750,104.667,-178.5409,-0.2387,0.0000
C01788=20.141,-117.557,104.133,-177.6257,-1.9629,0.0000
C01789=15.705,-110.997,103.471,-178.4754,-4.6328,0.0000
C01790=14.289,-102.010,102.199,-179.2658,-5.0011,0.0000
C01791=13.065,-92.111,99.556,-179.3173,-4.6124,0.0000
C01792=11.961,-83.022,95.993,-179.3784,-3.9245,0.0000
C01793=10.968,-76.031,92.442,-179.6279,-1.9440,0.0000
C01794=9.276,-71.863,89.838,166.8248,13.0264,0.0000
C01795=5.407,-70.720,88.800,149.0673,3.7344,0.0000
C01796=2.289,-70.783,88.755,148.0116,-1.3922,0.0000
C01797=0.000,-70.811,88.785,148.0029,-0.0009,0.0000
C01798=0.000,-70.811,88.785,148.0029,-0.0009,0.0000
C01799=-2.288,-70.783,88.755,148.0116,1.3932,0.0000
C01800=-5.408,-70.720,88.800,149.0681,-3.7371,0.0000
C01801=-9.276,-71.863,89.838,166.8255,-13.0263,0.0000
C01802=-10.968,-76.031,92.442,-179.6279,1.9440,0.0000
C01803=-11.961,-83.022,95.993,-179.3784,3.9245,0.0000
C01804=-13.065,-92.111,99.556,-179.3173,4.6124,0.0000
C01805=-14.289,-102.010,102.199,-179.2658,5.0011,0.0000
C01806=-15.705,-110.997,103.471,-178.4754,4.6328,0.0000
C01807=-20.141,-117.557,104.133,-177.6257,1.9629,0.0000
C01808=-27.134,-120.750,104.667,-178.5409,0.2387,0.0000
C01809=-35.236,-119.917,105.202,-179.9070,-0.0271,0.0000
C01810=-43.628,-117.138,105.553,-179.9895,-0.0039,0.0000
C01811=-51.979,-113.678,105.553,-179.9898,-0.0047,0.0000
C01812=-59.878,-109.710,105.202,-179.9151,-0.0466,0.0000
C01813=-66.196,-104.570,104.667,-179.1369,-1.2005,0.0000
C01814=-68.883,-97.367,104.133,-179.7087,-3.0654,0.0000
C01815=-67.381,-89.592,103.471,177.7964,-4.3530,0.0000
C01816=-62.028,-82.235,102.199,176.9767,-4.0577,0.0000
C01817=-55.894,-74.370,99.556,177.2164,-3.7459,0.0000
C01818=-50.248,-67.163,95.993,177.6615,-3.2156,0.0000
C01819=-46.007,-61.518,92.442,178.8881,-1.6378,0.0000
C01820=-44.256,-57.374,89.838,179.8891,18.2174,0.0000
C01821=-46.183,-53.830,88.800,159.3140,25.1687,0.0000
C01822=-48.433,-51.670,88.755,155.3527,22.9995,0.0000
C01823=-50.071,-50.071,88.785,156.1636,23.8353,0.0000
C01824=-51.669,-48.433,88.755,157.0010,24.6479,0.0000
C01825=-53.830,-46.183,88.800,154.8304,20.6837,0.0000
C01826=-57.374,-44.256,89.838,161.7832,0.1105,0.0000
C01827=-61.518,-46.007,92.442,-178.3622,1.1119,0.0000
C01828=-67.163,-50.248,95.993,-176.7844,2.3385,0.0000
C01829=-74.370,-55.894,99.556,-176.2541,2.7836,0.0000
C01830=-82.235,-62.028,102.199,-175.9423,3.0233,0.0000
C01831=-89.592,-67.381,103.471,-175.6470,2.2036,0.0000
C01832=-97.367,-68.883,104.133,-176.9346,-0.2913,0.0000
C01833=-104.570,-66.196,104.667,-178.7995,-0.8631,0.0000
C01834=-109.710,-59.878,105.202,-179.9534,-0.0849,0.0000
C01835=-113.678,-51.979,105.553,-179.9953,-0.0102,0.0000
C01836=-117.138,-43.628,105.553,-179.9961,-0.0105,0.0000
C01837=-119.917,-35.236,105.202,-179.9729,-0.0930,0.0000
C01838=-120.750,-27.134,104.667,179.7613,-1.4591,0.0000
C01839=-117.557,-20.141,104.133,178.0371,-2.3743,0.0000
C01840=-110.997,-15.705,103.471,175.3672,-1.5246,0.0000
C01841=-102.010,-14.289,102.199,174.9989,-0.7342,0.0000
C01842=-92.111,-13.065,99.556,175.3876,-0.6827,0.0000
C01843=-83.022,-11.961,95.993,176.0755,-0.6216,0.0000
C01844=-76.031,-10.968,92.442,178.0560,-0.3721,0.0000
C01845=-71.863,-9.276,89.838,-166.9736,13.1752,0.0000
C01846=-70.720,-5.407,88.800,-176.2656,30.9327,0.0000
C01847=-70.783,-2.289,88.755,178.6078,31.9884,0.0000
C01848=-70.811,0.000,88.785,179.9991,31.9971,0.0000
C01849=-70.783,2.288,88.755,-178.6068,31.9884,0.0000
C01850=-70.720,5.408,88.800,176.2629,30.9319,0.0000
C01851=-71.863,9.276,89.838,166.9737,13.1745,0.0000
C01852=-76.031,10.968,92.442,-178.0560,-0.3721,0.0000
C01853=-83.022,11.961,95.993,-176.0755,-0.6216,0.0000
C01854=-92.111,13.065,99.556,-175.3876,-0.6827,0.0000
C01855=-102.010,14.289,102.199,-174.9989,-0.7342,0.0000
C01856=-110.997,15.705,103.471,-175.3672,-1.5246,0.0000
C01857=-117.557,20.141,104.133,-178.0371,-2.3743,0.0000
C01858=-120.750,27.134,104.667,-179.7613,-1.4591,0.0000
